C01823=1018.796,230.980,371.499,168.951,51.014,159.703
C01824=1018.803,231.229,371.472,168.955,51.007,159.702
C01825=1018.808,231.478,371.446,168.959,51.001,159.701
C01826=1018.814,231.727,371.419,168.964,50.995,159.701
C01827=1018.820,231.975,371.392,168.967,50.989,159.700
C01828=1018.826,232.223,371.365,168.971,50.983,159.699
C01829=1018.832,232.472,371.338,168.976,50.976,159.699
C01830=1018.838,232.720,371.311,168.979,50.970,159.698
C01831=1018.844,232.969,371.285,168.984,50.964,159.698
C01832=1018.850,233.217,371.258,168.988,50.958,159.697
C01833=1018.856,233.444,371.234,168.992,50.952,159.697
C01834=1018.861,233.670,371.210,168.996,50.947,159.696
C01835=1018.867,233.895,371.185,169.000,50.941,159.695
C01836=1018.872,234.122,371.161,169.003,50.936,159.695
C01837=1018.877,234.348,371.136,169.007,50.930,159.694
C01838=1018.882,234.574,371.112,169.011,50.924,159.694
C01839=1018.888,234.800,371.087,169.015,50.919,159.693
C01840=1018.893,235.026,371.063,169.019,50.913,159.693
C01841=1018.900,235.275,371.036,169.022,50.907,159.692
C01842=1018.905,235.523,371.009,169.027,50.901,159.692
C01843=1018.911,235.771,370.982,169.031,50.895,159.691
C01844=1018.917,236.019,370.955,169.034,50.889,159.690
C01845=1018.924,236.268,370.928,169.040,50.883,159.690
C01846=1018.929,236.517,370.902,169.043,50.877,159.689
C01847=1018.936,236.766,370.875,169.047,50.871,159.688
C01848=1018.942,237.014,370.847,169.052,50.864,159.688
C01849=1018.948,237.262,370.821,169.056,50.859,159.687
C01850=1018.954,237.511,370.794,169.060,50.852,159.687
C01851=1018.960,237.759,370.766,169.064,50.846,159.686
C01852=1018.966,238.007,370.740,169.068,50.840,159.686
C01853=1018.972,238.256,370.713,169.073,50.834,159.685
C01854=1018.978,238.504,370.686,169.077,50.828,159.684
C01855=1018.985,238.753,370.658,169.080,50.822,159.684
C01856=1018.990,239.002,370.631,169.085,50.817,159.683
C01857=1018.996,239.249,370.604,169.089,50.810,159.683
C01858=1019.002,239.498,370.577,169.093,50.805,159.682
C01859=1019.008,239.747,370.550,169.098,50.799,159.682
C01860=1019.014,239.996,370.522,169.102,50.793,159.681
C01861=1019.020,240.244,370.495,169.106,50.787,159.681
C01862=1019.026,240.492,370.468,169.111,50.781,159.680
C01863=1019.032,240.740,370.439,169.114,50.775,159.680
C01864=1019.037,240.989,370.413,169.119,50.770,159.679
C01865=1019.044,241.237,370.385,169.123,50.764,159.678
C01866=1019.049,241.486,370.358,169.127,50.758,159.678
C01867=1019.056,241.734,370.330,169.131,50.752,159.677
C01868=1019.061,241.983,370.303,169.135,50.747,159.677
C01869=1019.067,242.231,370.275,169.140,50.741,159.676
C01870=1019.073,242.480,370.248,169.144,50.735,159.676
C01871=1019.079,242.728,370.220,169.148,50.730,159.675
C01872=1019.085,242.976,370.193,169.153,50.723,159.675
C01873=1019.091,243.225,370.166,169.157,50.718,159.674
C01874=1019.097,243.473,370.138,169.161,50.712,159.674
C01875=1019.102,243.721,370.110,169.165,50.707,159.673
C01876=1019.109,243.970,370.082,169.170,50.701,159.673
C01877=1019.114,244.218,370.054,169.174,50.695,159.672
C01878=1019.121,244.467,370.027,169.178,50.690,159.672
C01879=1019.126,244.715,369.999,169.182,50.684,159.671
C01880=1019.132,244.964,369.971,169.187,50.679,159.671
C01881=1019.138,245.211,369.943,169.191,50.673,159.670
C01882=1019.144,245.460,369.915,169.195,50.667,159.670
C01883=1019.149,245.708,369.887,169.199,50.662,159.669
C01884=1019.156,245.957,369.860,169.203,50.657,159.669
C01885=1019.161,246.205,369.832,169.208,50.651,159.669
C01886=1019.168,246.454,369.804,169.213,50.645,159.668
C01887=1019.174,246.703,369.776,169.217,50.640,159.668
C01888=1019.179,246.951,369.748,169.221,50.635,159.667
C01889=1019.186,247.199,369.720,169.226,50.628,159.667
C01890=1019.191,247.447,369.692,169.230,50.623,159.666
C01891=1019.197,247.696,369.664,169.234,50.618,159.666
C01892=1019.203,247.944,369.637,169.238,50.612,159.665
C01893=1019.208,248.167,369.611,169.242,50.608,159.665
C01894=1019.213,248.390,369.587,169.245,50.602,159.664
C01895=1019.219,248.612,369.562,169.250,50.598,159.664
C01896=1019.224,248.835,369.536,169.253,50.593,159.663
C01897=1019.230,249.058,369.511,169.258,50.588,159.663
C01898=1019.235,249.280,369.486,169.262,50.583,159.663
C01899=1019.241,249.504,369.461,169.265,50.578,159.662
C01900=1019.246,249.726,369.436,169.269,50.573,159.662
C01901=1019.252,249.975,369.408,169.273,50.568,159.661
C01902=1019.258,250.224,369.380,169.278,50.562,159.661
C01903=1019.264,250.472,369.352,169.282,50.557,159.660
C01904=1019.271,250.720,369.323,169.287,50.551,159.660
C01905=1019.276,250.968,369.295,169.291,50.546,159.660
C01906=1019.282,251.216,369.267,169.295,50.541,159.659
C01907=1019.288,251.465,369.239,169.300,50.536,159.659
C01908=1019.294,251.714,369.211,169.305,50.530,159.659
C01909=1019.300,251.962,369.183,169.309,50.525,159.658
C01910=1019.306,252.210,369.155,169.313,50.519,159.658
C01911=1019.312,252.459,369.127,169.317,50.514,159.657
C01912=1019.319,252.707,369.098,169.321,50.509,159.657
C01913=1019.325,252.955,369.070,169.326,50.503,159.656
C01914=1019.331,253.203,369.042,169.331,50.498,159.656
C01915=1019.337,253.452,369.014,169.335,50.493,159.656
C01916=1019.344,253.700,368.986,169.339,50.488,159.655
C01917=1019.350,253.949,368.957,169.343,50.482,159.655
C01918=1019.356,254.196,368.930,169.348,50.477,159.654
C01919=1019.362,254.445,368.902,169.352,50.471,159.654
C01920=1019.368,254.693,368.872,169.357,50.466,159.653
C01921=1019.375,254.942,368.845,169.361,50.461,159.653
C01922=1019.380,255.191,368.816,169.366,50.455,159.653
C01923=1019.386,255.439,368.788,169.370,50.450,159.652
C01924=1019.393,255.686,368.760,169.375,50.445,159.652
C01925=1019.399,255.935,368.732,169.379,50.440,159.651
C01926=1019.405,256.184,368.703,169.383,50.435,159.651
C01927=1019.412,256.432,368.675,169.388,50.429,159.650
C01928=1019.418,256.680,368.647,169.393,50.424,159.650
C01929=1019.423,256.929,368.619,169.397,50.419,159.650
C01930=1019.430,257.176,368.590,169.401,50.414,159.649
C01931=1019.436,257.425,368.562,169.406,50.409,159.649
C01932=1019.442,257.673,368.533,169.411,50.403,159.649
C01933=1019.449,257.922,368.505,169.415,50.398,159.648
C01934=1019.455,258.170,368.476,169.419,50.393,159.648
C01935=1019.461,258.419,368.448,169.423,50.388,159.647
C01936=1019.468,258.667,368.420,169.429,50.383,159.647
C01937=1019.474,258.915,368.391,169.433,50.378,159.647
C01938=1019.480,259.164,368.363,169.437,50.372,159.646
C01939=1019.487,259.412,368.334,169.442,50.368,159.646
C01940=1019.492,259.660,368.306,169.446,50.362,159.645
C01941=1019.498,259.908,368.277,169.451,50.357,159.645
C01942=1019.505,260.156,368.248,169.456,50.352,159.645
C01943=1019.511,260.405,368.220,169.460,50.347,159.645
C01944=1019.517,260.653,368.191,169.464,50.342,159.644
C01945=1019.523,260.901,368.162,169.469,50.337,159.644
C01946=1019.529,261.149,368.133,169.473,50.333,159.644
C01947=1019.535,261.398,368.104,169.477,50.327,159.643
C01948=1019.542,261.646,368.075,169.482,50.323,159.643
C01949=1019.548,261.894,368.046,169.487,50.318,159.643
C01950=1019.554,262.142,368.017,169.492,50.313,159.642
C01951=1019.560,262.390,367.988,169.496,50.308,159.642
C01952=1019.566,262.639,367.960,169.501,50.303,159.642
C01953=1019.571,262.861,367.934,169.504,50.299,159.641
C01954=1019.577,263.083,367.908,169.509,50.294,159.641
C01955=1019.582,263.305,367.882,169.513,50.290,159.641
C01956=1019.588,263.527,367.856,169.517,50.286,159.641
C01957=1019.593,263.749,367.830,169.521,50.281,159.640
C01958=1019.599,263.970,367.804,169.525,50.277,159.640
C01959=1019.605,264.192,367.778,169.529,50.272,159.639
C01960=1019.610,264.415,367.752,169.534,50.268,159.639
C01961=1019.616,264.663,367.723,169.538,50.263,159.639
C01962=1019.622,264.911,367.694,169.542,50.259,159.639
C01963=1019.629,265.159,367.665,169.547,50.254,159.638
C01964=1019.635,265.407,367.636,169.551,50.249,159.638
C01965=1019.640,265.656,367.606,169.556,50.245,159.638
C01966=1019.647,265.904,367.577,169.560,50.240,159.638
C01967=1019.653,266.152,367.548,169.566,50.235,159.637
C01968=1019.659,266.400,367.519,169.570,50.230,159.637
C01969=1019.665,266.648,367.490,169.575,50.226,159.637
C01970=1019.671,266.896,367.460,169.579,50.221,159.637
C01971=1019.678,267.145,367.430,169.584,50.216,159.636
C01972=1019.684,267.393,367.401,169.589,50.212,159.636
C01973=1019.691,267.641,367.372,169.593,50.207,159.636
C01974=1019.696,267.890,367.343,169.598,50.202,159.635
C01975=1019.702,268.138,367.314,169.602,50.198,159.635
C01976=1019.709,268.385,367.284,169.607,50.193,159.635
C01977=1019.714,268.634,367.254,169.612,50.188,159.635
C01978=1019.721,268.882,367.225,169.617,50.183,159.634
C01979=1019.727,269.131,367.196,169.621,50.179,159.634
C01980=1019.734,269.379,367.167,169.626,50.174,159.634
C01981=1019.740,269.627,367.136,169.630,50.170,159.634
C01982=1019.746,269.875,367.107,169.635,50.165,159.633
C01983=1019.751,270.123,367.078,169.639,50.160,159.633
C01984=1019.758,270.371,367.048,169.644,50.156,159.633
C01985=1019.765,270.619,367.019,169.649,50.152,159.633
C01986=1019.770,270.867,366.988,169.653,50.147,159.632
C01987=1019.777,271.115,366.959,169.658,50.142,159.632
C01988=1019.782,271.364,366.930,169.662,50.138,159.632
C01989=1019.789,271.611,366.900,169.668,50.133,159.632
C01990=1019.796,271.860,366.870,169.673,50.129,159.632
C01991=1019.801,272.108,366.840,169.677,50.124,159.631
C01992=1019.808,272.356,366.811,169.682,50.120,159.631
C01993=1019.814,272.604,366.781,169.687,50.116,159.631
C01994=1019.820,272.853,366.751,169.691,50.111,159.631
C01995=1019.826,273.101,366.721,169.696,50.106,159.630
C01996=1019.832,273.349,366.692,169.701,50.102,159.630
C01997=1019.838,273.597,366.661,169.705,50.098,159.630
C01998=1019.845,273.845,366.632,169.710,50.093,159.630
C01999=1019.851,274.093,366.602,169.715,50.089,159.630
C02000=1019.857,274.341,366.572,169.719,50.085,159.629
C02001=1019.864,274.590,366.542,169.724,50.081,159.629
C02002=1019.870,274.837,366.512,169.729,50.076,159.629
C02003=1019.876,275.086,366.483,169.733,50.071,159.629
C02004=1019.882,275.333,366.453,169.739,50.067,159.629
C02005=1019.889,275.582,366.422,169.744,50.062,159.628
C02006=1019.895,275.830,366.393,169.749,50.058,159.628
C02007=1019.901,276.078,366.363,169.753,50.054,159.628
C02008=1019.907,276.326,366.332,169.758,50.050,159.628
C02009=1019.914,276.574,366.302,169.763,50.045,159.628
C02010=1019.920,276.823,366.272,169.768,50.041,159.628
C02011=1019.926,277.071,366.242,169.772,50.037,159.627
C02012=1019.932,277.318,366.212,169.777,50.033,159.627
C02013=1019.938,277.542,366.184,169.781,50.029,159.627
C02014=1019.943,277.767,366.157,169.786,50.025,159.627
C02015=1019.949,277.991,366.130,169.790,50.021,159.627
C02016=1019.955,278.215,366.102,169.795,50.017,159.627
C02017=1019.960,278.440,366.075,169.799,50.014,159.627
C02018=1019.966,278.664,366.047,169.804,50.010,159.626
C02019=1019.971,278.888,366.020,169.808,50.006,159.626
C02020=1019.977,279.112,365.993,169.813,50.002,159.626
C02021=1019.983,279.361,365.962,169.817,49.998,159.626
C02022=1019.990,279.608,365.932,169.822,49.994,159.626
C02023=1019.996,279.857,365.901,169.827,49.990,159.626
C02024=1020.002,280.105,365.871,169.832,49.986,159.626
C02025=1020.008,280.353,365.840,169.837,49.982,159.626
C02026=1020.014,280.601,365.810,169.841,49.977,159.625
C02027=1020.021,280.849,365.780,169.846,49.973,159.625
C02028=1020.027,281.097,365.750,169.851,49.969,159.625
C02029=1020.033,281.345,365.719,169.856,49.965,159.625
C02030=1020.039,281.593,365.689,169.861,49.961,159.625
C02031=1020.046,281.841,365.659,169.866,49.957,159.625
C02032=1020.053,282.089,365.627,169.870,49.953,159.625
C02033=1020.058,282.337,365.597,169.875,49.949,159.624
C02034=1020.065,282.585,365.566,169.880,49.945,159.624
C02035=1020.071,282.834,365.536,169.885,49.941,159.624
C02036=1020.078,283.081,365.506,169.890,49.937,159.624
C02037=1020.084,283.330,365.475,169.895,49.933,159.624
C02038=1020.090,283.577,365.444,169.900,49.929,159.624
C02039=1020.097,283.825,365.413,169.906,49.924,159.624
C02040=1020.103,284.073,365.384,169.910,49.920,159.624
C02041=1020.110,284.321,365.353,169.915,49.916,159.624
C02042=1020.117,284.569,365.321,169.920,49.912,159.624
C02043=1020.122,284.817,365.291,169.925,49.909,159.623
C02044=1020.129,285.066,365.260,169.930,49.905,159.623
C02045=1020.135,285.313,365.229,169.935,49.901,159.623
C02046=1020.141,285.561,365.199,169.940,49.897,159.623
C02047=1020.147,285.809,365.167,169.945,49.893,159.623
C02048=1020.154,286.057,365.137,169.950,49.889,159.623
C02049=1020.161,286.305,365.105,169.955,49.886,159.623
C02050=1020.166,286.553,365.075,169.960,49.882,159.623
C02051=1020.173,286.801,365.044,169.965,49.878,159.623
C02052=1020.180,287.049,365.013,169.970,49.874,159.623
C02053=1020.186,287.296,364.982,169.975,49.870,159.623
C02054=1020.192,287.545,364.951,169.980,49.866,159.623
C02055=1020.199,287.793,364.920,169.985,49.863,159.623
C02056=1020.205,288.041,364.889,169.990,49.859,159.623
C02057=1020.211,288.289,364.858,169.995,49.855,159.623
C02058=1020.218,288.537,364.827,170.000,49.851,159.623
C02059=1020.224,288.784,364.796,170.005,49.847,159.623
C02060=1020.231,289.032,364.765,170.010,49.844,159.623
C02061=1020.237,289.281,364.734,170.015,49.840,159.622
C02062=1020.244,289.529,364.702,170.020,49.836,159.623
C02063=1020.250,289.776,364.671,170.025,49.832,159.622
C02064=1020.256,290.025,364.640,170.031,49.828,159.622
C02065=1020.262,290.273,364.609,170.036,49.824,159.622
C02066=1020.269,290.521,364.577,170.041,49.821,159.622
C02067=1020.275,290.768,364.546,170.046,49.817,159.622
C02068=1020.282,291.016,364.515,170.052,49.814,159.622
C02069=1020.288,291.264,364.484,170.057,49.810,159.622
C02070=1020.295,291.512,364.453,170.061,49.806,159.622
C02071=1020.302,291.760,364.421,170.067,49.803,159.622
C02072=1020.307,292.007,364.389,170.072,49.799,159.622
C02073=1020.314,292.238,364.361,170.076,49.796,159.622
C02074=1020.320,292.469,364.331,170.081,49.792,159.622
C02075=1020.325,292.699,364.302,170.086,49.788,159.622
C02076=1020.332,292.929,364.273,170.091,49.786,159.622
C02077=1020.338,293.160,364.243,170.096,49.782,159.622
C02078=1020.343,293.390,364.214,170.101,49.778,159.622
C02079=1020.349,293.620,364.185,170.105,49.775,159.622
C02080=1020.355,293.851,364.155,170.110,49.772,159.623
C02081=1020.361,294.098,364.123,170.116,49.769,159.623
C02082=1020.367,294.346,364.092,170.121,49.765,159.623
C02083=1020.373,294.595,364.060,170.126,49.762,159.623
C02084=1020.380,294.842,364.028,170.131,49.758,159.623
C02085=1020.386,295.090,363.996,170.136,49.755,159.623
C02086=1020.392,295.338,363.963,170.141,49.751,159.623
C02087=1020.399,295.585,363.932,170.147,49.748,159.623
C02088=1020.405,295.834,363.900,170.152,49.745,159.623
C02089=1020.412,296.081,363.868,170.157,49.741,159.623
C02090=1020.418,296.329,363.836,170.163,49.738,159.623
C02091=1020.424,296.577,363.805,170.168,49.734,159.623
C02092=1020.431,296.825,363.772,170.173,49.731,159.623
C02093=1020.437,297.073,363.740,170.178,49.728,159.623
C02094=1020.443,297.321,363.709,170.183,49.724,159.623
C02095=1020.450,297.568,363.676,170.189,49.721,159.623
C02096=1020.456,297.816,363.644,170.194,49.718,159.624
C02097=1020.462,298.064,363.612,170.199,49.714,159.623
C02098=1020.469,298.312,363.580,170.204,49.711,159.624
C02099=1020.475,298.560,363.548,170.210,49.707,159.624
C02100=1020.482,298.808,363.515,170.215,49.704,159.624
C02101=1020.488,299.055,363.484,170.220,49.701,159.624
C02102=1020.495,299.303,363.451,170.226,49.698,159.624
C02103=1020.501,299.551,363.420,170.231,49.694,159.624
C02104=1020.507,299.799,363.388,170.236,49.691,159.624
C02105=1020.514,300.047,363.355,170.241,49.688,159.624
C02106=1020.521,300.294,363.323,170.247,49.685,159.624
C02107=1020.527,300.542,363.291,170.252,49.681,159.624
C02108=1020.534,300.790,363.259,170.257,49.678,159.625
C02109=1020.540,301.038,363.227,170.263,49.675,159.625
C02110=1020.547,301.285,363.195,170.268,49.671,159.625
C02111=1020.553,301.533,363.163,170.273,49.668,159.625
C02112=1020.559,301.781,363.130,170.279,49.665,159.625
C02113=1020.567,302.029,363.097,170.284,49.662,159.625
C02114=1020.573,302.277,363.065,170.289,49.658,159.625
C02115=1020.580,302.524,363.033,170.295,49.656,159.625
C02116=1020.586,302.772,363.000,170.300,49.653,159.626
C02117=1020.592,303.020,362.968,170.305,49.649,159.626
C02118=1020.599,303.267,362.936,170.311,49.646,159.626
C02119=1020.606,303.516,362.903,170.317,49.642,159.626
C02120=1020.613,303.763,362.871,170.322,49.639,159.626
C02121=1020.619,304.011,362.839,170.328,49.637,159.626
C02122=1020.625,304.259,362.806,170.333,49.633,159.626
C02123=1020.632,304.506,362.774,170.339,49.630,159.627
C02124=1020.639,304.754,362.741,170.344,49.627,159.627
C02125=1020.646,305.002,362.709,170.349,49.624,159.627
C02126=1020.652,305.250,362.677,170.355,49.621,159.627
C02127=1020.658,305.497,362.644,170.360,49.618,159.627
C02128=1020.666,305.745,362.611,170.365,49.614,159.627
C02129=1020.672,305.993,362.579,170.371,49.612,159.628
C02130=1020.679,306.240,362.547,170.377,49.608,159.628
C02131=1020.686,306.489,362.513,170.383,49.605,159.628
C02132=1020.693,306.736,362.481,170.388,49.602,159.628
C02133=1020.699,306.976,362.450,170.394,49.599,159.628
C02134=1020.706,307.214,362.418,170.399,49.596,159.628
C02135=1020.712,307.454,362.387,170.404,49.594,159.628
C02136=1020.719,307.693,362.355,170.409,49.590,159.629
C02137=1020.725,307.932,362.324,170.415,49.588,159.629
C02138=1020.732,308.171,362.292,170.420,49.584,159.629
C02139=1020.739,308.410,362.261,170.426,49.582,159.629
C02140=1020.745,308.650,362.229,170.431,49.579,159.629
C02141=1020.752,308.897,362.196,170.437,49.576,159.630
C02142=1020.759,309.144,362.164,170.442,49.573,159.630
C02143=1020.766,309.393,362.131,170.447,49.569,159.630
C02144=1020.773,309.640,362.098,170.454,49.567,159.630
C02145=1020.780,309.888,362.065,170.459,49.563,159.630
C02146=1020.786,310.135,362.032,170.465,49.561,159.631
C02147=1020.792,310.383,361.999,170.470,49.558,159.631
C02148=1020.800,310.631,361.965,170.476,49.555,159.631
C02149=1020.806,310.878,361.933,170.481,49.552,159.631
C02150=1020.812,311.125,361.899,170.487,49.550,159.632
C02151=1020.819,311.374,361.865,170.493,49.547,159.632
C02152=1020.825,311.621,361.832,170.498,49.544,159.632
C02153=1020.832,311.869,361.799,170.504,49.542,159.632
C02154=1020.838,312.116,361.765,170.509,49.539,159.633
C02155=1020.845,312.365,361.732,170.515,49.536,159.633
C02156=1020.852,312.612,361.698,170.521,49.533,159.633
C02157=1020.858,312.859,361.665,170.526,49.531,159.633
C02158=1020.865,313.107,361.632,170.532,49.528,159.634
C02159=1020.871,313.354,361.598,170.538,49.526,159.634
C02160=1020.878,313.602,361.565,170.544,49.523,159.634
C02161=1020.884,313.849,361.531,170.550,49.520,159.635
C02162=1020.892,314.097,361.497,170.556,49.517,159.635
C02163=1020.898,314.345,361.463,170.561,49.515,159.635
C02164=1020.904,314.593,361.430,170.567,49.512,159.636
C02165=1020.912,314.840,361.396,170.573,49.510,159.636
C02166=1020.918,315.087,361.363,170.578,49.507,159.636
C02167=1020.924,315.336,361.329,170.584,49.504,159.636
C02168=1020.931,315.583,361.296,170.590,49.502,159.637
C02169=1020.938,315.831,361.262,170.595,49.499,159.637
C02170=1020.945,316.078,361.228,170.601,49.497,159.637
C02171=1020.951,316.325,361.194,170.608,49.494,159.638
C02172=1020.958,316.573,361.160,170.613,49.491,159.638
C02173=1020.965,316.821,361.127,170.619,49.488,159.638
C02174=1020.971,317.069,361.093,170.625,49.486,159.639
C02175=1020.978,317.316,361.059,170.630,49.483,159.639
C02176=1020.986,317.564,361.025,170.636,49.481,159.639
C02177=1020.992,317.811,360.992,170.642,49.478,159.639
C02178=1020.999,318.059,360.957,170.649,49.476,159.640
C02179=1021.006,318.307,360.924,170.655,49.473,159.640
C02180=1021.013,318.554,360.890,170.660,49.471,159.641
C02181=1021.020,318.801,360.856,170.666,49.468,159.641
C02182=1021.026,319.049,360.822,170.672,49.465,159.641
C02183=1021.033,319.297,360.788,170.678,49.463,159.642
C02184=1021.040,319.545,360.754,170.683,49.461,159.642
C02185=1021.046,319.792,360.720,170.690,49.458,159.642
C02186=1021.054,320.040,360.686,170.696,49.456,159.643
C02187=1021.061,320.287,360.653,170.702,49.453,159.643
C02188=1021.068,320.534,360.618,170.707,49.451,159.643
C02189=1021.075,320.782,360.584,170.713,49.448,159.644
C02190=1021.082,321.030,360.550,170.719,49.446,159.644
C02191=1021.088,321.277,360.516,170.726,49.443,159.644
C02192=1021.096,321.525,360.482,170.732,49.441,159.645
C02193=1021.102,321.767,360.449,170.737,49.439,159.645
C02194=1021.109,322.008,360.415,170.743,49.436,159.645
C02195=1021.116,322.250,360.382,170.749,49.434,159.646
C02196=1021.123,322.492,360.349,170.755,49.432,159.646
C02197=1021.130,322.733,360.315,170.761,49.430,159.647
C02198=1021.137,322.975,360.282,170.766,49.427,159.647
C02199=1021.144,323.217,360.249,170.772,49.425,159.647
C02200=1021.151,323.458,360.215,170.778,49.423,159.648
C02201=1021.158,323.706,360.181,170.785,49.420,159.648
C02202=1021.164,323.954,360.147,170.791,49.418,159.649
C02203=1021.172,324.201,360.112,170.797,49.416,159.649
C02204=1021.179,324.448,360.078,170.802,49.413,159.649
C02205=1021.186,324.696,360.043,170.809,49.411,159.650
C02206=1021.193,324.944,360.009,170.815,49.408,159.650
C02207=1021.201,325.192,359.975,170.821,49.406,159.651
C02208=1021.207,325.439,359.940,170.827,49.404,159.651
C02209=1021.215,325.687,359.906,170.834,49.401,159.652
C02210=1021.222,325.934,359.872,170.840,49.399,159.652
C02211=1021.229,326.182,359.838,170.846,49.397,159.652
C02212=1021.236,326.429,359.803,170.852,49.395,159.653
C02213=1021.244,326.676,359.768,170.859,49.393,159.653
C02214=1021.250,326.924,359.734,170.865,49.391,159.654
C02215=1021.258,327.171,359.699,170.870,49.388,159.654
C02216=1021.264,327.418,359.664,170.876,49.386,159.655
C02217=1021.272,327.667,359.629,170.882,49.384,159.655
C02218=1021.278,327.914,359.594,170.889,49.382,159.656
C02219=1021.286,328.162,359.560,170.895,49.380,159.656
C02220=1021.292,328.409,359.525,170.902,49.378,159.657
C02221=1021.299,328.656,359.489,170.908,49.376,159.657
C02222=1021.306,328.904,359.454,170.915,49.374,159.658
C02223=1021.313,329.151,359.420,170.921,49.372,159.658
C02224=1021.321,329.399,359.384,170.927,49.370,159.659
C02225=1021.328,329.646,359.349,170.933,49.368,159.659
C02226=1021.334,329.894,359.314,170.940,49.366,159.660
C02227=1021.342,330.141,359.280,170.946,49.364,159.660
C02228=1021.349,330.388,359.244,170.952,49.362,159.661
C02229=1021.356,330.636,359.209,170.958,49.360,159.661
C02230=1021.363,330.883,359.174,170.965,49.357,159.662
C02231=1021.370,331.130,359.139,170.971,49.355,159.662
C02232=1021.378,331.378,359.104,170.977,49.354,159.663
C02233=1021.384,331.626,359.069,170.983,49.352,159.663
C02234=1021.392,331.873,359.033,170.990,49.350,159.664
C02235=1021.399,332.120,358.998,170.996,49.348,159.664
C02236=1021.406,332.368,358.963,171.002,49.346,159.665
C02237=1021.413,332.615,358.928,171.009,49.344,159.665
C02238=1021.421,332.863,358.892,171.015,49.342,159.666
C02239=1021.428,333.110,358.857,171.022,49.340,159.666
C02240=1021.435,333.357,358.822,171.028,49.339,159.667
C02241=1021.442,333.605,358.786,171.035,49.336,159.668
C02242=1021.450,333.852,358.750,171.041,49.335,159.668
C02243=1021.456,334.099,358.715,171.047,49.333,159.669
C02244=1021.464,334.347,358.679,171.054,49.331,159.669
C02245=1021.471,334.594,358.644,171.061,49.329,159.670
C02246=1021.478,334.841,358.608,171.067,49.327,159.670
C02247=1021.485,335.089,358.572,171.074,49.326,159.671
C02248=1021.492,335.335,358.537,171.080,49.324,159.672
C02249=1021.500,335.584,358.501,171.087,49.322,159.672
C02250=1021.507,335.830,358.465,171.094,49.320,159.673
C02251=1021.514,336.078,358.430,171.100,49.319,159.674
C02252=1021.521,336.325,358.394,171.106,49.317,159.674
C02253=1021.528,336.565,358.358,171.112,49.316,159.675
C02254=1021.535,336.805,358.324,171.118,49.314,159.675
C02255=1021.542,337.044,358.289,171.126,49.312,159.676
C02256=1021.549,337.283,358.254,171.132,49.310,159.676
C02257=1021.556,337.523,358.220,171.138,49.309,159.677
C02258=1021.563,337.763,358.185,171.144,49.307,159.678
C02259=1021.570,338.002,358.151,171.151,49.305,159.678
C02260=1021.578,338.242,358.115,171.157,49.304,159.679
C02261=1021.585,338.488,358.080,171.164,49.302,159.679
C02262=1021.592,338.736,358.044,171.170,49.301,159.680
C02263=1021.599,338.983,358.008,171.178,49.299,159.681
C02264=1021.607,339.231,357.972,171.184,49.297,159.681
C02265=1021.615,339.478,357.936,171.190,49.296,159.682
C02266=1021.622,339.725,357.900,171.198,49.294,159.683
C02267=1021.629,339.972,357.864,171.204,49.293,159.683
C02268=1021.636,340.220,357.827,171.210,49.291,159.684
C02269=1021.643,340.467,357.791,171.218,49.290,159.685
C02270=1021.651,340.714,357.755,171.224,49.288,159.685
C02271=1021.659,340.962,357.719,171.231,49.286,159.686
C02272=1021.665,341.209,357.682,171.238,49.285,159.687
C02273=1021.673,341.456,357.646,171.244,49.283,159.687
C02274=1021.680,341.704,357.610,171.251,49.282,159.688
C02275=1021.688,341.950,357.573,171.258,49.280,159.689
C02276=1021.695,342.197,357.536,171.265,49.279,159.690
C02277=1021.702,342.445,357.500,171.271,49.277,159.690
C02278=1021.710,342.692,357.464,171.279,49.276,159.691
C02279=1021.717,342.940,357.427,171.285,49.274,159.692
C02280=1021.724,343.186,357.391,171.292,49.273,159.692
C02281=1021.732,343.434,357.354,171.299,49.271,159.693
C02282=1021.739,343.681,357.318,171.306,49.271,159.694
C02283=1021.747,343.928,357.281,171.313,49.269,159.695
C02284=1021.755,344.176,357.244,171.320,49.268,159.695
C02285=1021.762,344.423,357.207,171.327,49.266,159.696
C02286=1021.769,344.670,357.171,171.333,49.265,159.697
C02287=1021.777,344.917,357.135,171.341,49.263,159.698
C02288=1021.784,345.164,357.097,171.347,49.262,159.698
C02289=1021.792,345.412,357.061,171.354,49.261,159.699
C02290=1021.799,345.659,357.024,171.361,49.259,159.700
C02291=1021.806,345.906,356.987,171.368,49.258,159.701
C02292=1021.814,346.153,356.950,171.375,49.257,159.701
C02293=1021.822,346.400,356.913,171.382,49.256,159.702
C02294=1021.829,346.648,356.877,171.389,49.254,159.703
C02295=1021.837,346.894,356.840,171.396,49.253,159.704
C02296=1021.844,347.142,356.803,171.403,49.252,159.705
C02297=1021.852,347.389,356.766,171.411,49.251,159.705
C02298=1021.859,347.636,356.728,171.417,49.249,159.706
C02299=1021.867,347.883,356.692,171.425,49.248,159.707
C02300=1021.874,348.131,356.655,171.431,49.247,159.708
C02301=1021.882,348.378,356.618,171.439,49.245,159.708
C02302=1021.890,348.625,356.580,171.446,49.245,159.709
C02303=1021.898,348.871,356.543,171.453,49.244,159.710
C02304=1021.905,349.119,356.506,171.460,49.242,159.711
C02305=1021.912,349.366,356.468,171.467,49.241,159.712
C02306=1021.920,349.613,356.431,171.474,49.240,159.713
C02307=1021.927,349.860,356.394,171.482,49.239,159.714
C02308=1021.935,350.108,356.356,171.488,49.238,159.714
C02309=1021.943,350.354,356.319,171.496,49.237,159.715
C02310=1021.950,350.601,356.281,171.503,49.236,159.716
C02311=1021.958,350.848,356.245,171.510,49.235,159.717
C02312=1021.966,351.095,356.207,171.518,49.234,159.718
C02313=1021.973,351.333,356.171,171.524,49.232,159.719
C02314=1021.981,351.571,356.135,171.531,49.232,159.719
C02315=1021.988,351.809,356.098,171.539,49.231,159.720
C02316=1021.995,352.047,356.062,171.546,49.230,159.721
C02317=1022.003,352.286,356.026,171.552,49.229,159.722
C02318=1022.010,352.524,355.990,171.560,49.228,159.723
C02319=1022.018,352.761,355.954,171.566,49.227,159.724
C02320=1022.026,352.999,355.917,171.574,49.226,159.725
C02321=1022.033,353.246,355.880,171.581,49.225,159.726
C02322=1022.040,353.493,355.842,171.589,49.224,159.727
C02323=1022.049,353.740,355.804,171.596,49.222,159.727
C02324=1022.056,353.987,355.767,171.603,49.222,159.728
C02325=1022.064,354.234,355.729,171.610,49.221,159.729
C02326=1022.072,354.481,355.691,171.619,49.220,159.730
C02327=1022.080,354.728,355.653,171.625,49.220,159.731
C02328=1022.088,354.976,355.615,171.633,49.219,159.732
C02329=1022.095,355.222,355.577,171.641,49.218,159.733
C02330=1022.103,355.469,355.539,171.648,49.217,159.734
C02331=1022.111,355.716,355.501,171.655,49.216,159.735
C02332=1022.119,355.963,355.463,171.663,49.215,159.736
C02333=1022.127,356.210,355.425,171.670,49.215,159.737
C02334=1022.134,356.457,355.387,171.678,49.214,159.738
C02335=1022.142,356.704,355.349,171.686,49.213,159.739
C02336=1022.150,356.951,355.310,171.692,49.212,159.740
C02337=1022.158,357.198,355.273,171.700,49.211,159.741
C02338=1022.166,357.445,355.235,171.708,49.210,159.742
C02339=1022.174,357.692,355.196,171.716,49.209,159.743
C02340=1022.182,357.939,355.158,171.723,49.209,159.744
C02341=1022.190,358.186,355.119,171.731,49.208,159.745
C02342=1022.198,358.432,355.081,171.739,49.207,159.746
C02343=1022.206,358.680,355.042,171.747,49.207,159.747
C02344=1022.213,358.926,355.004,171.753,49.206,159.748
C02345=1022.221,359.173,354.965,171.761,49.206,159.749
C02346=1022.230,359.420,354.928,171.769,49.205,159.750
C02347=1022.238,359.667,354.889,171.777,49.204,159.751
C02348=1022.246,359.914,354.851,171.785,49.203,159.752
C02349=1022.254,360.161,354.812,171.792,49.203,159.753
C02350=1022.261,360.408,354.773,171.800,49.202,159.754
C02351=1022.269,360.655,354.735,171.808,49.201,159.755
C02352=1022.277,360.901,354.696,171.816,49.201,159.756
C02353=1022.285,361.148,354.657,171.823,49.200,159.757
C02354=1022.293,361.396,354.618,171.831,49.200,159.758
C02355=1022.301,361.642,354.579,171.839,49.199,159.759
C02356=1022.309,361.889,354.540,171.847,49.199,159.760
C02357=1022.317,362.136,354.502,171.855,49.199,159.762
C02358=1022.325,362.382,354.463,171.863,49.198,159.762
C02359=1022.333,362.629,354.424,171.870,49.197,159.764
C02360=1022.341,362.876,354.385,171.878,49.197,159.765
C02361=1022.349,363.123,354.346,171.886,49.197,159.766
C02362=1022.357,363.370,354.306,171.894,49.196,159.767
C02363=1022.365,363.617,354.268,171.902,49.196,159.768
C02364=1022.373,363.863,354.229,171.911,49.195,159.769
C02365=1022.381,364.110,354.190,171.919,49.195,159.770
C02366=1022.390,364.357,354.151,171.926,49.195,159.771
C02367=1022.398,364.604,354.111,171.934,49.194,159.773
C02368=1022.406,364.851,354.072,171.942,49.194,159.774
C02369=1022.414,365.098,354.033,171.950,49.193,159.775
C02370=1022.422,365.344,353.994,171.958,49.193,159.776
C02371=1022.431,365.592,353.955,171.966,49.192,159.777
C02372=1022.438,365.837,353.916,171.974,49.192,159.778
C02373=1022.447,366.079,353.877,171.982,49.192,159.779
C02374=1022.455,366.321,353.839,171.991,49.191,159.781
C02375=1022.463,366.562,353.800,171.999,49.191,159.782
C02376=1022.471,366.804,353.762,172.006,49.191,159.783
C02377=1022.479,367.044,353.723,172.014,49.190,159.784
C02378=1022.487,367.286,353.685,172.022,49.190,159.785
C02379=1022.495,367.528,353.646,172.030,49.190,159.786
C02380=1022.504,367.769,353.607,172.039,49.189,159.788
C02381=1022.512,368.015,353.568,172.047,49.189,159.789
C02382=1022.520,368.262,353.528,172.055,49.189,159.790
C02383=1022.529,368.509,353.489,172.063,49.189,159.791
C02384=1022.536,368.756,353.449,172.072,49.189,159.793
C02385=1022.545,369.002,353.410,172.080,49.188,159.794
C02386=1022.553,369.249,353.369,172.088,49.188,159.795
C02387=1022.562,369.496,353.329,172.096,49.188,159.796
C02388=1022.569,369.743,353.289,172.105,49.188,159.798
C02389=1022.578,369.989,353.249,172.113,49.188,159.799
C02390=1022.586,370.236,353.209,172.121,49.188,159.800
C02391=1022.594,370.482,353.170,172.130,49.188,159.801
C02392=1022.602,370.729,353.129,172.138,49.188,159.803
C02393=1022.612,370.976,353.090,172.146,49.188,159.804
C02394=1022.620,371.222,353.049,172.155,49.188,159.805
C02395=1022.628,371.469,353.010,172.164,49.187,159.806
C02396=1022.636,371.715,352.969,172.172,49.187,159.808
C02397=1022.645,371.962,352.929,172.181,49.187,159.809
C02398=1022.653,372.209,352.889,172.189,49.188,159.810
C02399=1022.662,372.455,352.849,172.197,49.187,159.812
C02400=1022.670,372.702,352.808,172.206,49.187,159.813
C02401=1022.679,372.948,352.768,172.214,49.187,159.814
C02402=1022.687,373.195,352.728,172.224,49.187,159.816
C02403=1022.696,373.442,352.688,172.232,49.187,159.817
C02404=1022.704,373.688,352.647,172.241,49.188,159.818
C02405=1022.713,373.935,352.607,172.249,49.188,159.820
C02406=1022.721,374.181,352.566,172.258,49.188,159.821
C02407=1022.730,374.427,352.526,172.267,49.188,159.823
C02408=1022.739,374.675,352.486,172.275,49.188,159.824
C02409=1022.747,374.921,352.446,172.284,49.188,159.825
C02410=1022.756,375.168,352.405,172.292,49.188,159.827
C02411=1022.765,375.414,352.365,172.302,49.188,159.828
C02412=1022.773,375.661,352.324,172.310,49.188,159.829
C02413=1022.783,375.907,352.284,172.319,49.188,159.831
C02414=1022.791,376.154,352.243,172.328,49.189,159.832
C02415=1022.799,376.401,352.202,172.337,49.189,159.834
C02416=1022.808,376.646,352.162,172.345,49.189,159.835
C02417=1022.817,376.893,352.120,172.354,49.189,159.836
C02418=1022.825,377.139,352.080,172.364,49.189,159.838
C02419=1022.834,377.386,352.039,172.372,49.189,159.839
C02420=1022.843,377.632,351.997,172.381,49.190,159.841
C02421=1022.851,377.879,351.956,172.390,49.190,159.842
C02422=1022.860,378.125,351.916,172.399,49.191,159.844
C02423=1022.869,378.372,351.874,172.408,49.191,159.845
C02424=1022.877,378.618,351.833,172.418,49.191,159.847
C02425=1022.886,378.864,351.792,172.426,49.191,159.848
C02426=1022.895,379.111,351.751,172.435,49.192,159.850
C02427=1022.903,379.357,351.709,172.444,49.192,159.851
C02428=1022.912,379.603,351.668,172.453,49.193,159.853
C02429=1022.921,379.850,351.627,172.462,49.193,159.854
C02430=1022.930,380.096,351.586,172.471,49.193,159.856
C02431=1022.938,380.342,351.544,172.480,49.194,159.857
C02432=1022.947,380.589,351.503,172.490,49.194,159.859
C02433=1022.957,380.847,351.460,172.500,49.195,159.860
C02434=1022.965,381.105,351.416,172.509,49.195,159.862
C02435=1022.975,381.364,351.373,172.519,49.196,159.864
C02436=1022.984,381.622,351.329,172.528,49.196,159.865
C02437=1022.993,381.868,351.288,172.538,49.197,159.867
C02438=1023.003,382.114,351.246,172.547,49.197,159.868
C02439=1023.012,382.360,351.205,172.557,49.198,159.870
C02440=1023.021,382.607,351.163,172.566,49.198,159.872
C02441=1023.030,382.853,351.121,172.575,49.199,159.873
C02442=1023.039,383.100,351.080,172.584,49.200,159.875
C02443=1023.048,383.346,351.038,172.594,49.200,159.876
C02444=1023.056,383.592,350.996,172.603,49.201,159.878
C02445=1023.066,383.838,350.955,172.613,49.201,159.880
C02446=1023.075,384.085,350.913,172.623,49.201,159.881
C02447=1023.084,384.331,350.872,172.631,49.202,159.883
C02448=1023.093,384.577,350.830,172.641,49.202,159.884
C02449=1023.102,384.823,350.787,172.650,49.203,159.886
C02450=1023.111,385.070,350.746,172.660,49.204,159.888
C02451=1023.120,385.316,350.704,172.670,49.204,159.889
C02452=1023.130,385.562,350.661,172.679,49.205,159.891
C02453=1023.140,385.808,350.620,172.689,49.206,159.893
C02454=1023.149,386.055,350.578,172.699,49.207,159.894
C02455=1023.157,386.301,350.535,172.708,49.207,159.896
C02456=1023.166,386.547,350.494,172.718,49.208,159.898
C02457=1023.175,386.793,350.451,172.728,49.209,159.899
C02458=1023.185,387.039,350.408,172.737,49.210,159.901
C02459=1023.194,387.286,350.367,172.747,49.210,159.903
C02460=1023.203,387.531,350.324,172.757,49.211,159.905
C02461=1023.212,387.777,350.282,172.767,49.212,159.906
C02462=1023.221,388.025,350.239,172.776,49.213,159.908
C02463=1023.230,388.270,350.197,172.786,49.214,159.910
C02464=1023.240,388.517,350.154,172.796,49.215,159.912
C02465=1023.250,388.763,350.111,172.806,49.215,159.913
C02466=1023.259,389.008,350.069,172.816,49.216,159.915
C02467=1023.269,389.255,350.026,172.825,49.217,159.917
C02468=1023.277,389.501,349.983,172.836,49.218,159.919
C02469=1023.286,389.747,349.941,172.846,49.219,159.921
C02470=1023.296,389.993,349.898,172.856,49.220,159.922
C02471=1023.305,390.239,349.855,172.866,49.221,159.924
C02472=1023.315,390.485,349.812,172.876,49.221,159.926
C02473=1023.324,390.731,349.770,172.885,49.223,159.928
C02474=1023.334,390.978,349.727,172.896,49.224,159.930
C02475=1023.342,391.223,349.683,172.906,49.225,159.932
C02476=1023.352,391.470,349.640,172.916,49.226,159.933
C02477=1023.362,391.715,349.598,172.926,49.227,159.935
C02478=1023.371,391.961,349.554,172.936,49.228,159.937
C02479=1023.381,392.208,349.511,172.947,49.229,159.939
C02480=1023.390,392.454,349.469,172.957,49.230,159.941
C02481=1023.400,392.699,349.425,172.967,49.231,159.943
C02482=1023.409,392.946,349.382,172.977,49.232,159.945
C02483=1023.419,393.191,349.339,172.988,49.233,159.946
C02484=1023.428,393.438,349.295,172.998,49.235,159.948
C02485=1023.438,393.684,349.252,173.008,49.236,159.950
C02486=1023.447,393.929,349.208,173.019,49.237,159.952
C02487=1023.457,394.176,349.165,173.029,49.238,159.954
C02488=1023.467,394.422,349.122,173.039,49.239,159.956
C02489=1023.476,394.668,349.077,173.050,49.241,159.958
C02490=1023.486,394.913,349.034,173.060,49.242,159.960
C02491=1023.495,395.159,348.990,173.071,49.243,159.962
C02492=1023.505,395.405,348.947,173.081,49.244,159.964
C02493=1023.516,395.700,348.895,173.094,49.246,159.966
C02494=1023.528,395.995,348.842,173.107,49.247,159.969
C02495=1023.540,396.289,348.790,173.120,49.249,159.971
C02496=1023.552,396.585,348.737,173.133,49.250,159.974
C02497=1023.561,396.830,348.693,173.143,49.252,159.976
C02498=1023.571,397.076,348.649,173.154,49.253,159.978
C02499=1023.580,397.322,348.605,173.164,49.255,159.980
C02500=1023.591,397.568,348.562,173.175,49.256,159.982
C02501=1023.600,397.814,348.518,173.186,49.257,159.984
C02502=1023.610,398.060,348.474,173.197,49.258,159.986
C02503=1023.620,398.306,348.429,173.207,49.260,159.988
C02504=1023.631,398.552,348.385,173.218,49.262,159.990
C02505=1023.640,398.798,348.341,173.230,49.263,159.992
C02506=1023.650,399.044,348.297,173.240,49.264,159.994
C02507=1023.660,399.289,348.252,173.251,49.266,159.996
C02508=1023.670,399.535,348.208,173.262,49.267,159.998
C02509=1023.679,399.781,348.163,173.273,49.269,160.001
C02510=1023.690,400.026,348.119,173.284,49.270,160.003
C02511=1023.700,400.273,348.075,173.295,49.272,160.005
C02512=1023.710,400.518,348.030,173.306,49.274,160.007
C02513=1023.720,400.763,347.986,173.318,49.275,160.009
C02514=1023.730,401.009,347.941,173.328,49.276,160.011
C02515=1023.740,401.256,347.896,173.340,49.278,160.014
C02516=1023.749,401.501,347.852,173.351,49.279,160.016
C02517=1023.759,401.747,347.807,173.362,49.281,160.018
C02518=1023.770,401.992,347.763,173.374,49.283,160.020
C02519=1023.780,402.238,347.717,173.384,49.285,160.022
C02520=1023.790,402.484,347.672,173.396,49.286,160.025
C02521=1023.800,402.729,347.627,173.407,49.288,160.027
C02522=1023.810,402.975,347.582,173.419,49.290,160.029
C02523=1023.820,403.220,347.537,173.430,49.291,160.031
C02524=1023.830,403.467,347.492,173.442,49.293,160.034
C02525=1023.840,403.712,347.447,173.454,49.295,160.036
C02526=1023.850,403.958,347.401,173.464,49.297,160.038
C02527=1023.861,404.203,347.357,173.476,49.299,160.040
C02528=1023.871,404.449,347.312,173.487,49.301,160.043
C02529=1023.881,404.694,347.266,173.499,49.302,160.045
C02530=1023.891,404.940,347.221,173.511,49.304,160.047
C02531=1023.902,405.186,347.175,173.522,49.306,160.050
C02532=1023.912,405.431,347.130,173.534,49.308,160.052
C02533=1023.922,405.677,347.084,173.546,49.309,160.054
C02534=1023.933,405.923,347.039,173.558,49.311,160.057
C02535=1023.943,406.168,346.994,173.569,49.314,160.059
C02536=1023.954,406.413,346.948,173.581,49.315,160.061
C02537=1023.964,406.660,346.903,173.593,49.317,160.064
C02538=1023.975,406.905,346.857,173.605,49.319,160.066
C02539=1023.985,407.150,346.812,173.617,49.321,160.069
C02540=1023.996,407.396,346.766,173.628,49.323,160.071
C02541=1024.006,407.641,346.720,173.640,49.325,160.073
C02542=1024.017,407.887,346.674,173.652,49.327,160.076
C02543=1024.027,408.133,346.629,173.665,49.329,160.078
C02544=1024.039,408.378,346.583,173.677,49.331,160.081
C02545=1024.049,408.624,346.537,173.689,49.333,160.083
C02546=1024.060,408.869,346.492,173.701,49.335,160.086
C02547=1024.071,409.114,346.445,173.713,49.337,160.088
C02548=1024.081,409.360,346.399,173.725,49.339,160.091
C02549=1024.092,409.606,346.353,173.738,49.341,160.093
C02550=1024.103,409.851,346.307,173.750,49.343,160.096
C02551=1024.113,410.097,346.260,173.762,49.346,160.098
C02552=1024.123,410.342,346.214,173.775,49.348,160.101
C02553=1024.136,410.634,346.160,173.789,49.350,160.104
C02554=1024.148,410.925,346.104,173.803,49.353,160.107
C02555=1024.162,411.217,346.049,173.818,49.356,160.110
C02556=1024.174,411.508,345.993,173.833,49.358,160.113
C02557=1024.185,411.753,345.947,173.846,49.360,160.116
C02558=1024.196,411.999,345.900,173.858,49.363,160.118
C02559=1024.207,412.244,345.854,173.871,49.365,160.121
C02560=1024.218,412.489,345.807,173.884,49.367,160.124
C02561=1024.229,412.761,345.756,173.898,49.370,160.126
C02562=1024.242,413.032,345.704,173.912,49.373,160.129
C02563=1024.254,413.303,345.652,173.925,49.375,160.132
C02564=1024.267,413.575,345.600,173.939,49.378,160.135
C02565=1024.277,413.820,345.553,173.953,49.380,160.138
C02566=1024.288,414.065,345.506,173.965,49.383,160.141
C02567=1024.300,414.311,345.459,173.978,49.385,160.143
C02568=1024.310,414.556,345.412,173.991,49.387,160.146
C02569=1024.321,414.802,345.365,174.004,49.390,160.149
C02570=1024.333,415.047,345.318,174.017,49.392,160.151
C02571=1024.344,415.292,345.271,174.030,49.394,160.154
C02572=1024.356,415.537,345.224,174.044,49.397,160.157
C02573=1024.366,415.783,345.176,174.056,49.400,160.160
C02574=1024.378,416.028,345.129,174.069,49.402,160.163
C02575=1024.388,416.274,345.081,174.083,49.405,160.165
C02576=1024.400,416.518,345.034,174.095,49.407,160.168
C02577=1024.410,416.764,344.986,174.109,49.410,160.171
C02578=1024.422,417.009,344.938,174.123,49.412,160.174
C02579=1024.433,417.254,344.891,174.136,49.415,160.177
C02580=1024.445,417.499,344.843,174.149,49.418,160.180
C02581=1024.456,417.744,344.796,174.162,49.420,160.183
C02582=1024.467,417.990,344.748,174.176,49.423,160.185
C02583=1024.479,418.235,344.700,174.190,49.426,160.188
C02584=1024.490,418.480,344.652,174.202,49.428,160.191
C02585=1024.501,418.725,344.604,174.217,49.431,160.194
C02586=1024.512,418.970,344.556,174.230,49.434,160.197
C02587=1024.524,419.215,344.508,174.244,49.436,160.200
C02588=1024.535,419.460,344.460,174.257,49.439,160.203
C02589=1024.547,419.705,344.412,174.271,49.442,160.206
C02590=1024.559,419.950,344.363,174.285,49.445,160.209
C02591=1024.570,420.195,344.315,174.299,49.448,160.212
C02592=1024.582,420.441,344.267,174.313,49.450,160.215
C02593=1024.593,420.686,344.219,174.327,49.453,160.218
C02594=1024.605,420.930,344.170,174.341,49.456,160.221
C02595=1024.617,421.176,344.122,174.354,49.459,160.224
C02596=1024.629,421.421,344.073,174.368,49.462,160.227
C02597=1024.641,421.666,344.026,174.382,49.465,160.230
C02598=1024.652,421.911,343.977,174.396,49.468,160.233
C02599=1024.664,422.156,343.929,174.410,49.471,160.236
C02600=1024.676,422.401,343.880,174.426,49.474,160.240
C02601=1024.687,422.646,343.831,174.440,49.476,160.243
C02602=1024.699,422.891,343.782,174.454,49.479,160.246
C02603=1024.711,423.136,343.733,174.468,49.483,160.249
C02604=1024.723,423.381,343.684,174.482,49.486,160.252
C02605=1024.734,423.625,343.635,174.496,49.488,160.255
C02606=1024.747,423.870,343.586,174.511,49.492,160.258
C02607=1024.758,424.115,343.537,174.526,49.495,160.262
C02608=1024.770,424.361,343.488,174.540,49.498,160.265
C02609=1024.782,424.605,343.439,174.555,49.501,160.268
C02610=1024.794,424.851,343.390,174.569,49.504,160.271
C02611=1024.806,425.095,343.341,174.584,49.507,160.275
C02612=1024.818,425.340,343.291,174.599,49.510,160.278
C02613=1024.835,425.669,343.225,174.619,49.515,160.282
C02614=1024.851,425.998,343.159,174.638,49.519,160.287
C02615=1024.867,426.325,343.092,174.658,49.523,160.291
C02616=1024.883,426.653,343.025,174.679,49.528,160.296
C02617=1024.896,426.899,342.976,174.693,49.531,160.299
C02618=1024.908,427.143,342.926,174.709,49.534,160.302
C02619=1024.920,427.387,342.876,174.724,49.537,160.306
C02620=1024.932,427.632,342.826,174.739,49.541,160.309
C02621=1024.944,427.877,342.776,174.754,49.544,160.313
C02622=1024.957,428.122,342.726,174.769,49.548,160.316
C02623=1024.969,428.367,342.676,174.785,49.551,160.320
C02624=1024.981,428.612,342.626,174.800,49.554,160.323
C02625=1024.993,428.856,342.576,174.815,49.558,160.326
C02626=1025.005,429.101,342.526,174.831,49.561,160.330
C02627=1025.018,429.345,342.476,174.846,49.565,160.334
C02628=1025.030,429.590,342.425,174.862,49.568,160.337
C02629=1025.043,429.835,342.375,174.878,49.571,160.341
C02630=1025.055,430.080,342.324,174.893,49.575,160.344
C02631=1025.069,430.324,342.274,174.908,49.579,160.348
C02632=1025.081,430.569,342.224,174.924,49.582,160.351
C02633=1025.094,430.813,342.173,174.940,49.586,160.355
C02634=1025.106,431.058,342.123,174.956,49.590,160.359
C02635=1025.119,431.303,342.072,174.972,49.593,160.362
C02636=1025.132,431.547,342.021,174.988,49.597,160.366
C02637=1025.144,431.792,341.971,175.004,49.600,160.369
C02638=1025.157,432.036,341.920,175.020,49.604,160.373
C02639=1025.170,432.281,341.869,175.037,49.607,160.377
C02640=1025.183,432.525,341.818,175.053,49.611,160.380
C02641=1025.196,432.770,341.767,175.069,49.615,160.384
C02642=1025.208,433.014,341.716,175.085,49.619,160.388
C02643=1025.222,433.259,341.665,175.101,49.622,160.392
C02644=1025.234,433.503,341.614,175.118,49.626,160.395
C02645=1025.248,433.747,341.562,175.134,49.630,160.399
C02646=1025.260,433.992,341.512,175.150,49.634,160.403
C02647=1025.274,434.236,341.460,175.168,49.637,160.407
C02648=1025.287,434.480,341.409,175.184,49.641,160.411
C02649=1025.300,434.725,341.358,175.201,49.645,160.415
C02650=1025.313,434.970,341.305,175.217,49.649,160.418
C02651=1025.325,435.214,341.254,175.234,49.652,160.422
C02652=1025.339,435.458,341.203,175.251,49.656,160.426
C02653=1025.352,435.702,341.151,175.268,49.660,160.430
C02654=1025.365,435.946,341.099,175.285,49.664,160.434
C02655=1025.378,436.191,341.047,175.302,49.668,160.438
C02656=1025.391,436.435,340.995,175.318,49.672,160.442
C02657=1025.405,436.680,340.944,175.336,49.676,160.446
C02658=1025.418,436.924,340.892,175.353,49.680,160.450
C02659=1025.432,437.168,340.839,175.371,49.684,160.454
C02660=1025.445,437.412,340.787,175.387,49.689,160.458
C02661=1025.458,437.656,340.735,175.405,49.692,160.462
C02662=1025.472,437.901,340.683,175.422,49.696,160.466
C02663=1025.485,438.145,340.631,175.440,49.700,160.470
C02664=1025.499,438.389,340.578,175.457,49.704,160.474
C02665=1025.512,438.633,340.526,175.475,49.708,160.478
C02666=1025.526,438.877,340.473,175.493,49.712,160.482
C02667=1025.539,439.121,340.421,175.511,49.717,160.487
C02668=1025.552,439.365,340.368,175.528,49.721,160.491
C02669=1025.567,439.610,340.315,175.546,49.725,160.495
C02670=1025.581,439.853,340.263,175.564,49.730,160.499
C02671=1025.594,440.098,340.210,175.581,49.734,160.503
C02672=1025.607,440.341,340.157,175.600,49.738,160.508
C02673=1025.620,440.553,340.111,175.615,49.741,160.511
C02674=1025.632,440.764,340.066,175.631,49.745,160.515
C02675=1025.644,440.976,340.020,175.647,49.749,160.519
C02676=1025.655,441.187,339.973,175.663,49.753,160.522
C02677=1025.668,441.398,339.927,175.679,49.756,160.526
C02678=1025.680,441.609,339.882,175.695,49.760,160.530
C02679=1025.692,441.820,339.836,175.710,49.764,160.534
C02680=1025.704,442.032,339.790,175.726,49.768,160.537
C02681=1025.718,442.275,339.736,175.746,49.772,160.542
C02682=1025.732,442.518,339.683,175.764,49.777,160.546
C02683=1025.747,442.761,339.631,175.782,49.781,160.551
C02684=1025.762,443.005,339.578,175.801,49.785,160.555
C02685=1025.778,443.248,339.527,175.819,49.789,160.559
C02686=1025.794,443.492,339.475,175.838,49.794,160.564
C02687=1025.810,443.735,339.424,175.857,49.798,160.568
C02688=1025.827,443.979,339.373,175.877,49.801,160.572
C02689=1025.844,444.222,339.323,175.896,49.805,160.577
C02690=1025.862,444.467,339.272,175.915,49.809,160.581
C02691=1025.880,444.711,339.223,175.935,49.813,160.586
C02692=1025.899,444.955,339.174,175.954,49.817,160.590
C02693=1025.918,445.199,339.125,175.973,49.820,160.594
C02694=1025.937,445.443,339.076,175.993,49.823,160.599
C02695=1025.957,445.687,339.028,176.013,49.827,160.603
C02696=1025.978,445.931,338.981,176.033,49.830,160.607
C02697=1025.999,446.176,338.933,176.053,49.834,160.612
C02698=1026.020,446.420,338.887,176.072,49.837,160.616
C02699=1026.042,446.665,338.840,176.092,49.840,160.620
C02700=1026.065,446.910,338.794,176.113,49.843,160.624
C02701=1026.087,447.154,338.748,176.132,49.847,160.629
C02702=1026.110,447.399,338.703,176.153,49.849,160.633
C02703=1026.134,447.644,338.657,176.172,49.852,160.637
C02704=1026.158,447.889,338.613,176.193,49.855,160.642
C02705=1026.183,448.133,338.569,176.214,49.858,160.646
C02706=1026.207,448.378,338.525,176.235,49.861,160.650
C02707=1026.233,448.624,338.482,176.255,49.864,160.655
C02708=1026.258,448.868,338.439,176.276,49.866,160.659
C02709=1026.284,449.113,338.396,176.297,49.869,160.663
C02710=1026.312,449.358,338.354,176.318,49.872,160.668
C02711=1026.340,449.604,338.312,176.339,49.874,160.672
C02712=1026.367,449.849,338.271,176.361,49.876,160.676
C02713=1026.395,450.095,338.230,176.381,49.879,160.680
C02714=1026.423,450.340,338.189,176.402,49.881,160.684
C02715=1026.452,450.585,338.149,176.424,49.883,160.689
C02716=1026.482,450.831,338.109,176.446,49.886,160.693
C02717=1026.512,451.076,338.069,176.468,49.887,160.697
C02718=1026.543,451.322,338.030,176.489,49.889,160.702
C02719=1026.573,451.567,337.991,176.511,49.892,160.706
C02720=1026.605,451.812,337.953,176.533,49.893,160.710
C02721=1026.637,452.059,337.916,176.555,49.895,160.714
C02722=1026.669,452.305,337.877,176.577,49.897,160.719
C02723=1026.702,452.550,337.840,176.600,49.899,160.723
C02724=1026.734,452.795,337.804,176.622,49.901,160.727
C02725=1026.769,453.041,337.768,176.644,49.903,160.732
C02726=1026.803,453.287,337.731,176.667,49.904,160.736
C02727=1026.838,453.533,337.696,176.689,49.906,160.740
C02728=1026.872,453.778,337.660,176.711,49.908,160.744
C02729=1026.908,454.024,337.626,176.735,49.909,160.749
C02730=1026.944,454.271,337.591,176.757,49.910,160.753
C02731=1026.981,454.516,337.558,176.780,49.912,160.757
C02732=1027.017,454.762,337.524,176.803,49.913,160.762
C02733=1026.744,454.840,337.186,176.805,49.972,160.781
C02734=1026.707,454.594,337.219,176.783,49.971,160.777
C02735=1026.671,454.349,337.252,176.760,49.970,160.772
C02736=1026.635,454.103,337.287,176.736,49.968,160.768
C02737=1026.599,453.856,337.322,176.714,49.967,160.764
C02738=1026.564,453.611,337.357,176.691,49.966,160.760
C02739=1026.529,453.366,337.392,176.668,49.964,160.755
C02740=1026.495,453.119,337.428,176.646,49.962,160.751
C02741=1026.461,452.873,337.464,176.624,49.961,160.747
C02742=1026.428,452.628,337.501,176.601,49.959,160.742
C02743=1026.395,452.382,337.537,176.579,49.957,160.738
C02744=1026.363,452.137,337.575,176.556,49.956,160.734
C02745=1026.330,451.890,337.613,176.534,49.954,160.730
C02746=1026.299,451.645,337.651,176.513,49.952,160.725
C02747=1026.268,451.401,337.689,176.490,49.950,160.721
C02748=1026.237,451.154,337.729,176.469,49.948,160.717
C02749=1026.207,450.909,337.768,176.447,49.946,160.713
C02750=1026.177,450.664,337.808,176.425,49.944,160.708
C02751=1026.148,450.418,337.847,176.404,49.942,160.704
C02752=1026.119,450.173,337.888,176.382,49.940,160.700
C02753=1026.091,449.927,337.929,176.361,49.938,160.696
C02754=1026.063,449.682,337.970,176.340,49.935,160.691
C02755=1026.035,449.437,338.012,176.319,49.933,160.687
C02756=1026.009,449.192,338.054,176.298,49.931,160.683
C02757=1025.982,448.947,338.096,176.277,49.928,160.678
C02758=1025.956,448.701,338.140,176.256,49.925,160.674
C02759=1025.930,448.456,338.183,176.235,49.923,160.670
C02760=1025.905,448.211,338.226,176.214,49.921,160.666
C02761=1025.881,447.967,338.271,176.194,49.918,160.661
C02762=1025.856,447.722,338.314,176.173,49.915,160.657
C02763=1025.833,447.477,338.360,176.152,49.912,160.653
C02764=1025.809,447.232,338.405,176.133,49.909,160.648
C02765=1025.786,446.987,338.450,176.112,49.906,160.644
C02766=1025.764,446.743,338.496,176.091,49.903,160.640
C02767=1025.742,446.498,338.543,176.072,49.900,160.636
C02768=1025.721,446.254,338.589,176.052,49.897,160.631
C02769=1025.699,446.009,338.636,176.032,49.894,160.627
C02770=1025.678,445.765,338.683,176.012,49.890,160.622
C02771=1025.658,445.520,338.732,175.992,49.887,160.618
C02772=1025.638,445.276,338.779,175.972,49.884,160.614
C02773=1025.619,445.032,338.828,175.953,49.880,160.610
C02774=1025.600,444.788,338.877,175.933,49.877,160.605
C02775=1025.582,444.544,338.927,175.914,49.874,160.601
C02776=1025.564,444.301,338.976,175.895,49.870,160.597
C02777=1025.546,444.056,339.027,175.876,49.865,160.592
C02778=1025.530,443.812,339.077,175.856,49.862,160.588
C02779=1025.513,443.569,339.128,175.837,49.858,160.584
C02780=1025.496,443.325,339.179,175.818,49.854,160.579
C02781=1025.480,443.082,339.231,175.799,49.850,160.575
C02782=1025.466,442.838,339.283,175.780,49.846,160.570
C02783=1025.450,442.595,339.336,175.762,49.842,160.566
C02784=1025.436,442.352,339.388,175.744,49.838,160.562
C02785=1025.422,442.109,339.442,175.725,49.834,160.557
C02786=1025.410,441.901,339.487,175.709,49.830,160.554
C02787=1025.398,441.694,339.532,175.694,49.827,160.550
C02788=1025.386,441.488,339.577,175.678,49.822,160.546
C02789=1025.374,441.280,339.622,175.662,49.819,160.543
C02790=1025.362,441.073,339.667,175.646,49.815,160.539
C02791=1025.351,440.866,339.713,175.631,49.812,160.535
C02792=1025.339,440.659,339.757,175.615,49.809,160.532
C02793=1025.327,440.452,339.803,175.601,49.805,160.528
C02794=1025.314,440.208,339.855,175.583,49.800,160.524
C02795=1025.300,439.964,339.907,175.564,49.797,160.520
C02796=1025.286,439.721,339.960,175.546,49.792,160.515
C02797=1025.272,439.476,340.014,175.528,49.788,160.511
C02798=1025.259,439.232,340.066,175.511,49.784,160.507
C02799=1025.245,438.988,340.118,175.493,49.780,160.503
C02800=1025.232,438.744,340.171,175.475,49.776,160.499
C02801=1025.218,438.500,340.223,175.458,49.772,160.495
C02802=1025.205,438.256,340.276,175.440,49.768,160.491
C02803=1025.192,438.011,340.328,175.423,49.764,160.486
C02804=1025.178,437.766,340.380,175.405,49.760,160.482
C02805=1025.164,437.523,340.433,175.387,49.756,160.478
C02806=1025.150,437.279,340.485,175.370,49.752,160.474
C02807=1025.137,437.035,340.536,175.352,49.748,160.470
C02808=1025.124,436.791,340.588,175.335,49.745,160.466
C02809=1025.111,436.546,340.641,175.319,49.740,160.462
C02810=1025.097,436.302,340.693,175.301,49.737,160.458
C02811=1025.084,436.058,340.745,175.284,49.733,160.454
C02812=1025.070,435.813,340.797,175.267,49.729,160.450
C02813=1025.058,435.569,340.847,175.250,49.725,160.447
C02814=1025.045,435.324,340.900,175.233,49.722,160.443
C02815=1025.031,435.080,340.952,175.217,49.718,160.439
C02816=1025.018,434.835,341.003,175.200,49.714,160.435
C02817=1025.005,434.592,341.054,175.183,49.710,160.431
C02818=1024.992,434.347,341.106,175.166,49.707,160.427
C02819=1024.979,434.103,341.157,175.150,49.703,160.423
C02820=1024.966,433.858,341.208,175.133,49.699,160.420
C02821=1024.953,433.614,341.259,175.116,49.695,160.416
C02822=1024.941,433.370,341.312,175.100,49.692,160.412
C02823=1024.928,433.125,341.362,175.083,49.688,160.408
C02824=1024.915,432.880,341.414,175.067,49.685,160.405
C02825=1024.902,432.636,341.464,175.051,49.681,160.401
C02826=1024.889,432.391,341.516,175.034,49.678,160.397
C02827=1024.876,432.147,341.566,175.018,49.674,160.393
C02828=1024.863,431.903,341.616,175.002,49.670,160.390
C02829=1024.850,431.658,341.667,174.986,49.667,160.386
C02830=1024.837,431.413,341.718,174.971,49.663,160.383
C02831=1024.825,431.169,341.769,174.955,49.660,160.379
C02832=1024.812,430.924,341.819,174.938,49.657,160.375
C02833=1024.799,430.680,341.870,174.922,49.653,160.372
C02834=1024.787,430.435,341.920,174.906,49.650,160.368
C02835=1024.774,430.191,341.971,174.890,49.646,160.365
C02836=1024.762,429.946,342.021,174.876,49.642,160.361
C02837=1024.749,429.702,342.072,174.860,49.639,160.357
C02838=1024.736,429.457,342.121,174.844,49.636,160.354
C02839=1024.724,429.212,342.171,174.828,49.633,160.350
C02840=1024.712,428.967,342.221,174.813,49.629,160.347
C02841=1024.699,428.723,342.272,174.797,49.626,160.344
C02842=1024.687,428.478,342.322,174.781,49.623,160.340
C02843=1024.674,428.234,342.372,174.767,49.619,160.337
C02844=1024.662,427.989,342.423,174.751,49.616,160.333
C02845=1024.650,427.744,342.473,174.736,49.613,160.330
C02846=1024.638,427.499,342.522,174.721,49.609,160.326
C02847=1024.626,427.254,342.572,174.706,49.607,160.323
C02848=1024.614,427.009,342.622,174.690,49.603,160.319
C02849=1024.601,426.765,342.672,174.675,49.600,160.316
C02850=1024.586,426.434,342.738,174.655,49.595,160.312
C02851=1024.569,426.104,342.806,174.634,49.592,160.307
C02852=1024.552,425.773,342.872,174.614,49.587,160.303
C02853=1024.536,425.441,342.940,174.595,49.583,160.298
C02854=1024.524,425.197,342.989,174.580,49.580,160.295
C02855=1024.512,424.952,343.038,174.565,49.577,160.292
C02856=1024.500,424.707,343.087,174.551,49.574,160.289
C02857=1024.488,424.462,343.136,174.536,49.571,160.285
C02858=1024.476,424.217,343.185,174.521,49.568,160.282
C02859=1024.464,423.973,343.235,174.507,49.565,160.279
C02860=1024.452,423.728,343.283,174.492,49.562,160.276
C02861=1024.440,423.483,343.333,174.478,49.558,160.272
C02862=1024.429,423.238,343.382,174.463,49.556,160.269
C02863=1024.417,422.993,343.430,174.449,49.553,160.266
C02864=1024.405,422.747,343.479,174.434,49.550,160.263
C02865=1024.393,422.503,343.528,174.420,49.547,160.260
C02866=1024.381,422.258,343.576,174.406,49.544,160.257
C02867=1024.369,422.013,343.626,174.392,49.541,160.254
C02868=1024.358,421.767,343.674,174.378,49.538,160.251
C02869=1024.346,421.523,343.722,174.363,49.536,160.247
C02870=1024.335,421.278,343.771,174.349,49.533,160.244
C02871=1024.323,421.033,343.819,174.335,49.530,160.241
C02872=1024.311,420.787,343.868,174.321,49.527,160.238
C02873=1024.299,420.542,343.916,174.307,49.525,160.235
C02874=1024.288,420.297,343.965,174.293,49.522,160.232
C02875=1024.276,420.052,344.012,174.280,49.519,160.229
C02876=1024.265,419.807,344.061,174.266,49.517,160.226
C02877=1024.253,419.562,344.108,174.252,49.514,160.223
C02878=1024.242,419.317,344.157,174.239,49.511,160.220
C02879=1024.230,419.071,344.204,174.224,49.509,160.217
C02880=1024.218,418.826,344.252,174.211,49.506,160.215
C02881=1024.207,418.581,344.300,174.197,49.503,160.211
C02882=1024.195,418.336,344.348,174.184,49.501,160.209
C02883=1024.185,418.091,344.396,174.170,49.498,160.206
C02884=1024.173,417.846,344.444,174.156,49.495,160.203
C02885=1024.162,417.601,344.492,174.143,49.493,160.200
C02886=1024.150,417.356,344.540,174.130,49.490,160.197
C02887=1024.139,417.110,344.587,174.116,49.488,160.194
C02888=1024.128,416.866,344.634,174.103,49.485,160.192
C02889=1024.117,416.620,344.683,174.090,49.483,160.189
C02890=1024.105,416.374,344.730,174.076,49.481,160.186
C02891=1024.095,416.130,344.778,174.063,49.478,160.183
C02892=1024.083,415.884,344.825,174.050,49.476,160.180
C02893=1024.073,415.640,344.873,174.037,49.473,160.177
C02894=1024.061,415.394,344.920,174.023,49.471,160.175
C02895=1024.050,415.148,344.967,174.011,49.468,160.172
C02896=1024.039,414.903,345.013,173.997,49.466,160.169
C02897=1024.028,414.658,345.062,173.985,49.463,160.166
C02898=1024.016,414.412,345.109,173.971,49.462,160.164
C02899=1024.005,414.167,345.155,173.959,49.459,160.161
C02900=1023.994,413.921,345.202,173.946,49.457,160.158
C02901=1023.984,413.676,345.249,173.933,49.454,160.156
C02902=1023.973,413.431,345.296,173.920,49.452,160.153
C02903=1023.961,413.186,345.343,173.908,49.449,160.150
C02904=1023.950,412.941,345.390,173.894,49.448,160.148
C02905=1023.940,412.695,345.435,173.882,49.445,160.145
C02906=1023.929,412.449,345.483,173.870,49.443,160.142
C02907=1023.918,412.204,345.530,173.856,49.441,160.140
C02908=1023.907,411.959,345.576,173.844,49.439,160.137
C02909=1023.896,411.713,345.623,173.831,49.436,160.134
C02910=1023.882,411.394,345.684,173.815,49.434,160.131
C02911=1023.867,411.074,345.744,173.798,49.431,160.128
C02912=1023.854,410.755,345.805,173.782,49.428,160.124
C02913=1023.840,410.434,345.865,173.766,49.425,160.121
C02914=1023.830,410.189,345.911,173.754,49.423,160.118
C02915=1023.819,409.944,345.957,173.741,49.421,160.116
C02916=1023.808,409.699,346.004,173.729,49.419,160.114
C02917=1023.798,409.453,346.050,173.717,49.417,160.111
C02918=1023.787,409.207,346.096,173.705,49.415,160.108
C02919=1023.776,408.962,346.142,173.693,49.413,160.106
C02920=1023.765,408.716,346.188,173.681,49.411,160.103
C02921=1023.755,408.471,346.234,173.669,49.410,160.101
C02922=1023.744,408.225,346.279,173.656,49.407,160.099
C02923=1023.734,407.979,346.325,173.644,49.406,160.096
C02924=1023.723,407.734,346.371,173.632,49.403,160.094
C02925=1023.712,407.488,346.417,173.620,49.402,160.091
C02926=1023.701,407.243,346.462,173.608,49.400,160.089
C02927=1023.691,406.998,346.508,173.596,49.398,160.086
C02928=1023.681,406.752,346.553,173.584,49.396,160.084
C02929=1023.670,406.506,346.599,173.573,49.394,160.082
C02930=1023.659,406.261,346.645,173.561,49.393,160.079
C02931=1023.650,406.015,346.690,173.549,49.390,160.077
C02932=1023.639,405.770,346.736,173.537,49.389,160.075
C02933=1023.628,405.524,346.782,173.525,49.387,160.072
C02934=1023.619,405.278,346.826,173.513,49.385,160.070
C02935=1023.607,405.033,346.872,173.502,49.383,160.068
C02936=1023.597,404.787,346.917,173.490,49.382,160.065
C02937=1023.587,404.541,346.962,173.478,49.380,160.063
C02938=1023.570,404.134,347.038,173.459,49.377,160.059
C02939=1023.553,403.727,347.112,173.441,49.374,160.055
C02940=1023.537,403.320,347.187,173.421,49.372,160.052
C02941=1023.520,402.913,347.261,173.402,49.369,160.048
C02942=1023.509,402.668,347.307,173.390,49.368,160.046
C02943=1023.499,402.422,347.352,173.380,49.366,160.043
C02944=1023.490,402.177,347.396,173.368,49.365,160.041
C02945=1023.479,401.930,347.442,173.357,49.362,160.039
C02946=1023.470,401.685,347.486,173.345,49.361,160.037
C02947=1023.459,401.440,347.531,173.335,49.359,160.035
C02948=1023.450,401.194,347.575,173.323,49.358,160.032
C02949=1023.440,400.947,347.620,173.312,49.356,160.030
C02950=1023.430,400.702,347.665,173.300,49.355,160.028
C02951=1023.419,400.457,347.709,173.290,49.354,160.026
C02952=1023.410,400.211,347.754,173.278,49.352,160.024
C02953=1023.400,399.964,347.798,173.267,49.350,160.022
C02954=1023.389,399.719,347.842,173.256,49.349,160.020
C02955=1023.379,399.474,347.887,173.245,49.348,160.017
C02956=1023.370,399.227,347.931,173.235,49.346,160.015
C02957=1023.360,398.982,347.976,173.223,49.345,160.013
C02958=1023.350,398.736,348.020,173.213,49.344,160.011
C02959=1023.341,398.490,348.064,173.202,49.342,160.009
C02960=1023.330,398.245,348.108,173.190,49.341,160.007
C02961=1023.321,397.999,348.152,173.180,49.340,160.005
C02962=1023.311,397.753,348.196,173.169,49.338,160.003
C02963=1023.301,397.507,348.241,173.158,49.337,160.001
C02964=1023.291,397.261,348.284,173.147,49.336,159.999
C02965=1023.281,397.015,348.328,173.137,49.334,159.997
C02966=1023.266,396.633,348.397,173.120,49.333,159.994
C02967=1023.250,396.252,348.464,173.103,49.330,159.990
C02968=1023.236,395.870,348.532,173.086,49.329,159.987
C02969=1023.221,395.488,348.600,173.071,49.327,159.984
C02970=1023.211,395.243,348.643,173.059,49.326,159.982
C02971=1023.202,394.997,348.687,173.049,49.325,159.980
C02972=1023.192,394.751,348.731,173.038,49.323,159.978
C02973=1023.182,394.505,348.774,173.028,49.322,159.976
C02974=1023.172,394.259,348.818,173.018,49.322,159.975
C02975=1023.163,394.014,348.861,173.007,49.320,159.973
C02976=1023.153,393.767,348.905,172.997,49.319,159.971
C02977=1023.144,393.521,348.948,172.987,49.318,159.969
C02978=1023.135,393.276,348.992,172.975,49.317,159.967
C02979=1023.125,393.029,349.034,172.965,49.316,159.965
C02980=1023.116,392.783,349.078,172.955,49.315,159.963
C02981=1023.106,392.537,349.121,172.945,49.314,159.961
C02982=1023.096,392.291,349.164,172.934,49.313,159.959
C02983=1023.086,392.045,349.207,172.924,49.312,159.957
C02984=1023.078,391.799,349.250,172.914,49.311,159.955
C02985=1023.068,391.553,349.294,172.904,49.310,159.954
C02986=1023.058,391.307,349.336,172.893,49.309,159.952
C02987=1023.049,391.061,349.380,172.883,49.308,159.950
C02988=1023.040,390.815,349.422,172.873,49.307,159.948
C02989=1023.030,390.569,349.465,172.863,49.306,159.946
C02990=1023.021,390.323,349.508,172.853,49.306,159.945
C02991=1023.012,390.076,349.551,172.844,49.305,159.943
C02992=1023.002,389.831,349.594,172.834,49.304,159.941
C02993=1022.992,389.584,349.637,172.823,49.303,159.939
C02994=1022.983,389.339,349.679,172.813,49.302,159.937
C02995=1022.975,389.092,349.722,172.803,49.302,159.936
C02996=1022.965,388.846,349.765,172.793,49.301,159.934
C02997=1022.956,388.600,349.807,172.783,49.300,159.932
C02998=1022.947,388.354,349.849,172.773,49.299,159.930
C02999=1022.937,388.107,349.892,172.764,49.298,159.929
C03000=1022.928,387.861,349.935,172.754,49.297,159.927
C03001=1022.919,387.616,349.977,172.744,49.297,159.925
C03002=1022.910,387.369,350.019,172.734,49.296,159.923
C03003=1022.900,387.123,350.062,172.724,49.296,159.922
C03004=1022.891,386.877,350.104,172.715,49.295,159.920
C03005=1022.882,386.631,350.146,172.705,49.294,159.918
C03006=1022.872,386.384,350.189,172.695,49.294,159.917
C03007=1022.863,386.138,350.230,172.685,49.293,159.915
C03008=1022.854,385.892,350.273,172.676,49.292,159.913
C03009=1022.845,385.646,350.315,172.666,49.292,159.912
C03010=1022.836,385.399,350.356,172.656,49.291,159.910
C03011=1022.827,385.154,350.399,172.646,49.290,159.908
C03012=1022.818,384.907,350.441,172.637,49.290,159.907
C03013=1022.809,384.660,350.482,172.628,49.289,159.905
C03014=1022.800,384.414,350.524,172.618,49.289,159.903
C03015=1022.790,384.168,350.567,172.609,49.288,159.902
C03016=1022.781,383.922,350.608,172.599,49.288,159.900
C03017=1022.772,383.676,350.649,172.589,49.287,159.898
C03018=1022.763,383.429,350.691,172.580,49.287,159.897
C03019=1022.754,383.183,350.733,172.571,49.286,159.895
C03020=1022.745,382.937,350.775,172.561,49.286,159.894
C03021=1022.736,382.690,350.816,172.552,49.285,159.892
C03022=1022.727,382.444,350.858,172.542,49.285,159.890
C03023=1022.718,382.198,350.900,172.534,49.285,159.889
C03024=1022.709,381.952,350.941,172.524,49.284,159.887
C03025=1022.700,381.705,350.983,172.515,49.284,159.886
C03026=1022.691,381.444,351.026,172.505,49.283,159.884
C03027=1022.681,381.184,351.070,172.495,49.283,159.883
C03028=1022.672,380.924,351.114,172.486,49.283,159.881
C03029=1022.662,380.664,351.157,172.476,49.282,159.879
C03030=1022.654,380.418,351.199,172.466,49.282,159.878
C03031=1022.645,380.171,351.240,172.457,49.282,159.876
C03032=1022.636,379.925,351.281,172.448,49.281,159.875
C03033=1022.627,379.678,351.323,172.439,49.281,159.873
C03034=1022.619,379.432,351.364,172.429,49.281,159.872
C03035=1022.609,379.186,351.405,172.421,49.281,159.870
C03036=1022.601,378.939,351.446,172.411,49.280,159.869
C03037=1022.592,378.693,351.488,172.403,49.280,159.867
C03038=1022.584,378.446,351.528,172.394,49.279,159.866
C03039=1022.575,378.200,351.570,172.384,49.280,159.864
C03040=1022.566,377.953,351.611,172.375,49.279,159.863
C03041=1022.558,377.707,351.652,172.366,49.279,159.861
C03042=1022.549,377.461,351.693,172.357,49.279,159.860
C03043=1022.541,377.214,351.733,172.349,49.278,159.858
C03044=1022.532,376.967,351.774,172.339,49.279,159.857
C03045=1022.524,376.722,351.816,172.331,49.278,159.856
C03046=1022.515,376.475,351.857,172.322,49.278,159.854
C03047=1022.506,376.228,351.897,172.312,49.278,159.853
C03048=1022.498,375.982,351.938,172.304,49.278,159.851
C03049=1022.488,375.735,351.978,172.295,49.278,159.850
C03050=1022.480,375.489,352.019,172.286,49.278,159.849
C03051=1022.472,375.242,352.060,172.278,49.278,159.847
C03052=1022.463,374.996,352.100,172.269,49.278,159.846
C03053=1022.454,374.749,352.141,172.260,49.278,159.844
C03054=1022.445,374.503,352.181,172.251,49.278,159.843
C03055=1022.437,374.255,352.221,172.243,49.278,159.842
C03056=1022.428,374.009,352.261,172.233,49.278,159.840
C03057=1022.420,373.762,352.302,172.225,49.278,159.839
C03058=1022.411,373.516,352.342,172.217,49.278,159.838
C03059=1022.403,373.269,352.382,172.208,49.278,159.836
C03060=1022.394,373.023,352.423,172.199,49.278,159.835
C03061=1022.386,372.776,352.463,172.190,49.278,159.834
C03062=1022.377,372.530,352.503,172.182,49.278,159.832
C03063=1022.369,372.283,352.544,172.174,49.278,159.831
C03064=1022.360,372.037,352.584,172.165,49.278,159.830
C03065=1022.352,371.790,352.623,172.156,49.278,159.828
C03066=1022.343,371.543,352.664,172.148,49.279,159.827
C03067=1022.335,371.296,352.704,172.139,49.279,159.826
C03068=1022.326,371.050,352.744,172.131,49.279,159.825
C03069=1022.319,370.803,352.784,172.123,49.279,159.823
C03070=1022.310,370.557,352.824,172.114,49.279,159.822
C03071=1022.302,370.310,352.864,172.105,49.280,159.821
C03072=1022.293,370.063,352.903,172.097,49.280,159.819
C03073=1022.285,369.817,352.944,172.089,49.280,159.818
C03074=1022.277,369.570,352.983,172.080,49.280,159.817
C03075=1022.269,369.323,353.023,172.072,49.280,159.816
C03076=1022.260,369.078,353.063,172.063,49.280,159.814
C03077=1022.252,368.831,353.103,172.055,49.281,159.813
C03078=1022.243,368.583,353.143,172.047,49.281,159.812
C03079=1022.236,368.336,353.183,172.039,49.281,159.811
C03080=1022.227,368.090,353.222,172.031,49.281,159.810
C03081=1022.219,367.843,353.261,172.022,49.282,159.808
C03082=1022.211,367.601,353.300,172.014,49.282,159.807
C03083=1022.202,367.359,353.339,172.006,49.282,159.806
C03084=1022.194,367.116,353.378,171.998,49.283,159.805
C03085=1022.186,366.874,353.417,171.990,49.283,159.804
C03086=1022.178,366.631,353.456,171.982,49.284,159.803
C03087=1022.169,366.389,353.494,171.974,49.284,159.801
C03088=1022.162,366.145,353.532,171.965,49.285,159.800
C03089=1022.154,365.903,353.571,171.957,49.285,159.799
C03090=1022.146,365.657,353.610,171.949,49.285,159.798
C03091=1022.137,365.410,353.650,171.941,49.286,159.797
C03092=1022.129,365.163,353.689,171.933,49.286,159.796
C03093=1022.121,364.916,353.728,171.925,49.287,159.794
C03094=1022.112,364.670,353.767,171.917,49.287,159.793
C03095=1022.105,364.423,353.807,171.909,49.288,159.792
C03096=1022.097,364.176,353.845,171.901,49.288,159.791
C03097=1022.089,363.930,353.884,171.893,49.289,159.790
C03098=1022.080,363.682,353.923,171.885,49.290,159.789
C03099=1022.072,363.436,353.962,171.877,49.290,159.788
C03100=1022.064,363.189,354.001,171.869,49.291,159.787
C03101=1022.055,362.942,354.040,171.861,49.291,159.785
C03102=1022.048,362.695,354.079,171.853,49.292,159.785
C03103=1022.040,362.449,354.119,171.845,49.293,159.783
C03104=1022.032,362.201,354.157,171.838,49.293,159.782
C03105=1022.024,361.954,354.196,171.829,49.293,159.781
C03106=1022.016,361.708,354.235,171.822,49.294,159.780
C03107=1022.008,361.461,354.273,171.814,49.295,159.779
C03108=1022.000,361.213,354.312,171.805,49.295,159.778
C03109=1021.992,360.968,354.351,171.798,49.296,159.777
C03110=1021.984,360.720,354.390,171.790,49.297,159.776
C03111=1021.976,360.473,354.429,171.783,49.297,159.775
C03112=1021.969,360.227,354.467,171.775,49.298,159.774
C03113=1021.960,359.980,354.506,171.767,49.299,159.773
C03114=1021.953,359.734,354.544,171.759,49.299,159.772
C03115=1021.944,359.486,354.583,171.751,49.300,159.771
C03116=1021.936,359.239,354.622,171.743,49.301,159.770
C03117=1021.929,358.993,354.660,171.735,49.302,159.769
C03118=1021.921,358.745,354.699,171.729,49.303,159.768
C03119=1021.913,358.499,354.737,171.720,49.303,159.767
C03120=1021.905,358.251,354.775,171.713,49.304,159.766
C03121=1021.898,358.005,354.813,171.705,49.305,159.765
C03122=1021.890,357.757,354.852,171.697,49.306,159.764
C03123=1021.881,357.511,354.889,171.690,49.306,159.763
C03124=1021.873,357.264,354.928,171.682,49.307,159.762
C03125=1021.866,357.017,354.965,171.675,49.308,159.761
C03126=1021.858,356.770,355.004,171.667,49.309,159.760
C03127=1021.850,356.523,355.042,171.659,49.310,159.759
C03128=1021.842,356.276,355.081,171.652,49.311,159.758
C03129=1021.834,356.029,355.118,171.644,49.312,159.757
C03130=1021.826,355.782,355.156,171.637,49.313,159.756
C03131=1021.818,355.535,355.195,171.629,49.314,159.755
C03132=1021.810,355.287,355.232,171.622,49.315,159.754
C03133=1021.803,355.041,355.271,171.614,49.316,159.753
C03134=1021.796,354.794,355.308,171.607,49.317,159.752
C03135=1021.787,354.547,355.346,171.599,49.318,159.751
C03136=1021.780,354.300,355.384,171.592,49.318,159.750
C03137=1021.772,354.053,355.422,171.584,49.319,159.749
C03138=1021.764,353.805,355.460,171.577,49.321,159.748
C03139=1021.756,353.559,355.497,171.570,49.321,159.748
C03140=1021.749,353.312,355.535,171.562,49.322,159.747
C03141=1021.740,353.064,355.572,171.555,49.324,159.746
C03142=1021.734,352.826,355.608,171.548,49.325,159.745
C03143=1021.726,352.587,355.646,171.540,49.326,159.744
C03144=1021.718,352.348,355.681,171.534,49.326,159.743
C03145=1021.711,352.109,355.718,171.526,49.328,159.742
C03146=1021.703,351.870,355.754,171.519,49.329,159.742
C03147=1021.696,351.631,355.791,171.512,49.330,159.741
C03148=1021.688,351.392,355.826,171.505,49.331,159.740
C03149=1021.681,351.152,355.863,171.498,49.332,159.739
C03150=1021.674,350.905,355.900,171.491,49.334,159.738
C03151=1021.666,350.658,355.937,171.483,49.335,159.737
C03152=1021.659,350.411,355.975,171.477,49.335,159.736
C03153=1021.650,350.164,356.012,171.469,49.337,159.736
C03154=1021.643,349.916,356.050,171.461,49.338,159.735
C03155=1021.635,349.669,356.087,171.455,49.339,159.734
C03156=1021.627,349.422,356.124,171.447,49.341,159.733
C03157=1021.620,349.175,356.162,171.440,49.342,159.732
C03158=1021.613,348.928,356.199,171.433,49.343,159.731
C03159=1021.605,348.681,356.236,171.425,49.344,159.731
C03160=1021.598,348.434,356.274,171.419,49.345,159.730
C03161=1021.590,348.187,356.311,171.412,49.347,159.729
C03162=1021.583,347.940,356.348,171.404,49.348,159.728
C03163=1021.575,347.693,356.384,171.398,49.349,159.727
C03164=1021.568,347.446,356.422,171.390,49.350,159.727
C03165=1021.560,347.199,356.459,171.383,49.352,159.726
C03166=1021.553,346.951,356.496,171.376,49.353,159.725
C03167=1021.545,346.704,356.533,171.370,49.355,159.724
C03168=1021.537,346.457,356.569,171.362,49.356,159.723
C03169=1021.530,346.210,356.606,171.355,49.357,159.723
C03170=1021.522,345.963,356.643,171.348,49.359,159.722
C03171=1021.515,345.715,356.680,171.341,49.360,159.721
C03172=1021.507,345.468,356.717,171.334,49.362,159.721
C03173=1021.499,345.221,356.753,171.327,49.363,159.720
C03174=1021.492,344.974,356.791,171.320,49.364,159.719
C03175=1021.485,344.727,356.827,171.313,49.366,159.718
C03176=1021.477,344.480,356.863,171.306,49.367,159.718
C03177=1021.470,344.232,356.900,171.299,49.369,159.717
C03178=1021.462,343.985,356.937,171.293,49.370,159.716
C03179=1021.454,343.738,356.973,171.285,49.372,159.715
C03180=1021.447,343.490,357.010,171.279,49.373,159.715
C03181=1021.440,343.244,357.046,171.272,49.375,159.714
C03182=1021.432,342.997,357.083,171.265,49.376,159.713
C03183=1021.425,342.749,357.120,171.258,49.378,159.712
C03184=1021.418,342.502,357.156,171.251,49.379,159.712
C03185=1021.410,342.254,357.192,171.244,49.381,159.711
C03186=1021.404,342.007,357.229,171.238,49.382,159.710
C03187=1021.396,341.760,357.266,171.230,49.384,159.710
C03188=1021.388,341.513,357.302,171.224,49.385,159.709
C03189=1021.381,341.266,357.338,171.217,49.388,159.708
C03190=1021.374,341.018,357.375,171.210,49.389,159.708
C03191=1021.366,340.771,357.411,171.203,49.391,159.707
C03192=1021.359,340.523,357.447,171.197,49.392,159.706
C03193=1021.352,340.277,357.483,171.189,49.394,159.706
C03194=1021.345,340.029,357.520,171.183,49.395,159.705
C03195=1021.338,339.782,357.555,171.176,49.397,159.704
C03196=1021.330,339.535,357.592,171.169,49.398,159.704
C03197=1021.322,339.287,357.628,171.163,49.400,159.703
C03198=1021.315,339.041,357.664,171.156,49.402,159.702
C03199=1021.308,338.792,357.699,171.150,49.403,159.702
C03200=1021.300,338.545,357.735,171.143,49.406,159.701
C03201=1021.293,338.298,357.771,171.136,49.407,159.700
C03202=1021.287,338.058,357.806,171.129,49.409,159.700
C03203=1021.279,337.817,357.841,171.123,49.411,159.699
C03204=1021.272,337.577,357.877,171.117,49.413,159.699
C03205=1021.265,337.336,357.911,171.110,49.414,159.698
C03206=1021.258,337.095,357.946,171.103,49.416,159.698
C03207=1021.250,336.854,357.981,171.097,49.418,159.697
C03208=1021.243,336.614,358.015,171.091,49.420,159.696
C03209=1021.237,336.373,358.050,171.085,49.421,159.696
C03210=1021.229,336.126,358.086,171.078,49.423,159.695
C03211=1021.222,335.879,358.122,171.071,49.425,159.694
C03212=1021.215,335.631,358.158,171.065,49.427,159.694
C03213=1021.208,335.384,358.193,171.058,49.429,159.693
C03214=1021.201,335.137,358.229,171.052,49.430,159.693
C03215=1021.193,334.889,358.264,171.045,49.432,159.692
C03216=1021.186,334.642,358.300,171.039,49.434,159.692
C03217=1021.179,334.394,358.336,171.032,49.436,159.691
C03218=1021.172,334.147,358.371,171.025,49.438,159.690
C03219=1021.165,333.900,358.407,171.019,49.440,159.690
C03220=1021.158,333.652,358.442,171.013,49.442,159.689
C03221=1021.151,333.405,358.478,171.006,49.444,159.689
C03222=1021.144,333.158,358.513,171.000,49.446,159.688
C03223=1021.137,332.910,358.549,170.994,49.448,159.688
C03224=1021.129,332.663,358.584,170.987,49.450,159.687
C03225=1021.122,332.416,358.619,170.981,49.452,159.687
C03226=1021.115,332.168,358.654,170.974,49.454,159.686
C03227=1021.108,331.921,358.690,170.968,49.456,159.686
C03228=1021.101,331.673,358.725,170.961,49.457,159.685
C03229=1021.093,331.425,358.760,170.954,49.460,159.684
C03230=1021.086,331.178,358.795,170.948,49.462,159.684
C03231=1021.079,330.931,358.831,170.942,49.464,159.683
C03232=1021.072,330.684,358.866,170.935,49.466,159.683
C03233=1021.064,330.436,358.901,170.929,49.468,159.682
C03234=1021.057,330.189,358.936,170.923,49.471,159.682
C03235=1021.051,329.942,358.971,170.916,49.473,159.682
C03236=1021.044,329.694,359.006,170.910,49.475,159.681
C03237=1021.036,329.446,359.040,170.904,49.477,159.681
C03238=1021.029,329.198,359.075,170.897,49.479,159.680
C03239=1021.023,328.951,359.111,170.891,49.481,159.680
C03240=1021.015,328.704,359.145,170.885,49.483,159.679
C03241=1021.008,328.457,359.180,170.878,49.485,159.678
C03242=1021.002,328.209,359.215,170.872,49.487,159.678
C03243=1020.995,327.962,359.250,170.867,49.490,159.678
C03244=1020.987,327.715,359.285,170.861,49.492,159.677
C03245=1020.980,327.466,359.320,170.853,49.494,159.677
C03246=1020.973,327.219,359.355,170.847,49.496,159.676
C03247=1020.967,326.971,359.390,170.842,49.499,159.676
C03248=1020.959,326.724,359.425,170.835,49.501,159.675
C03249=1020.953,326.476,359.459,170.829,49.503,159.675
C03250=1020.945,326.229,359.494,170.823,49.506,159.675
C03251=1020.938,325.982,359.527,170.816,49.508,159.674
C03252=1020.931,325.734,359.563,170.810,49.510,159.674
C03253=1020.924,325.487,359.596,170.804,49.512,159.673
C03254=1020.916,325.240,359.631,170.797,49.515,159.673
C03255=1020.909,324.992,359.665,170.792,49.517,159.672
C03256=1020.903,324.745,359.700,170.786,49.520,159.672
C03257=1020.895,324.497,359.734,170.779,49.522,159.672
C03258=1020.888,324.249,359.768,170.773,49.525,159.671
C03259=1020.881,324.002,359.803,170.767,49.527,159.671
C03260=1020.874,323.754,359.836,170.762,49.529,159.670
C03261=1020.867,323.506,359.870,170.755,49.532,159.670
C03262=1020.860,323.263,359.905,170.749,49.534,159.670
C03263=1020.853,323.021,359.938,170.743,49.537,159.669
C03264=1020.846,322.778,359.972,170.737,49.539,159.669
C03265=1020.839,322.535,360.004,170.732,49.542,159.669
C03266=1020.832,322.292,360.039,170.725,49.544,159.668
C03267=1020.825,322.050,360.072,170.719,49.546,159.668
C03268=1020.819,321.807,360.106,170.713,49.549,159.667
C03269=1020.812,321.564,360.138,170.708,49.552,159.667
C03270=1020.804,321.316,360.172,170.701,49.554,159.667
C03271=1020.798,321.069,360.207,170.695,49.557,159.666
C03272=1020.791,320.821,360.241,170.689,49.559,159.666
C03273=1020.783,320.574,360.275,170.684,49.562,159.666
C03274=1020.777,320.326,360.309,170.677,49.564,159.665
C03275=1020.770,320.079,360.343,170.671,49.567,159.665
C03276=1020.763,319.831,360.377,170.665,49.569,159.665
C03277=1020.756,319.583,360.411,170.659,49.572,159.664
C03278=1020.749,319.335,360.445,170.654,49.575,159.664
C03279=1020.743,319.088,360.479,170.647,49.577,159.664
C03280=1020.736,318.841,360.512,170.641,49.579,159.663
C03281=1020.728,318.593,360.546,170.635,49.582,159.663
C03282=1020.722,318.345,360.581,170.630,49.585,159.662
C03283=1020.715,318.098,360.614,170.624,49.587,159.662
C03284=1020.708,317.850,360.648,170.617,49.590,159.662
C03285=1020.702,317.602,360.682,170.612,49.593,159.662
C03286=1020.695,317.355,360.716,170.606,49.595,159.661
C03287=1020.688,317.108,360.750,170.600,49.598,159.661
C03288=1020.681,316.859,360.783,170.595,49.601,159.661
C03289=1020.675,316.612,360.817,170.588,49.604,159.660
C03290=1020.668,316.365,360.851,170.582,49.606,159.660
C03291=1020.661,316.117,360.884,170.577,49.609,159.660
C03292=1020.654,315.870,360.918,170.571,49.611,159.659
C03293=1020.648,315.622,360.952,170.565,49.614,159.659
C03294=1020.641,315.374,360.985,170.559,49.617,159.659
C03295=1020.634,315.127,361.019,170.553,49.620,159.658
C03296=1020.628,314.880,361.052,170.547,49.622,159.658
C03297=1020.621,314.631,361.086,170.542,49.626,159.658
C03298=1020.614,314.383,361.120,170.537,49.628,159.658
C03299=1020.608,314.136,361.153,170.531,49.631,159.657
C03300=1020.600,313.889,361.187,170.524,49.634,159.657
C03301=1020.595,313.641,361.220,170.519,49.636,159.657
C03302=1020.588,313.393,361.254,170.513,49.639,159.657
C03303=1020.581,313.146,361.287,170.507,49.642,159.656
C03304=1020.574,312.898,361.321,170.502,49.645,159.656
C03305=1020.568,312.651,361.355,170.496,49.647,159.656
C03306=1020.562,312.403,361.388,170.491,49.650,159.656
C03307=1020.555,312.155,361.421,170.484,49.653,159.655
C03308=1020.549,311.908,361.454,170.479,49.656,159.655
C03309=1020.541,311.660,361.488,170.473,49.659,159.655
C03310=1020.536,311.412,361.521,170.467,49.661,159.654
C03311=1020.529,311.165,361.555,170.462,49.665,159.654
C03312=1020.522,310.917,361.588,170.456,49.667,159.654
C03313=1020.516,310.670,361.621,170.451,49.670,159.654
C03314=1020.510,310.421,361.655,170.445,49.673,159.654
C03315=1020.503,310.174,361.689,170.440,49.676,159.653
C03316=1020.497,309.927,361.721,170.433,49.679,159.653
C03317=1020.489,309.679,361.754,170.428,49.682,159.653
C03318=1020.483,309.431,361.787,170.422,49.685,159.653
C03319=1020.476,309.184,361.819,170.417,49.688,159.653
C03320=1020.469,308.936,361.852,170.411,49.691,159.652
C03321=1020.462,308.688,361.885,170.405,49.695,159.652
C03322=1020.456,308.447,361.917,170.399,49.697,159.652
C03323=1020.450,308.208,361.948,170.394,49.701,159.652
C03324=1020.442,307.967,361.980,170.389,49.703,159.652
C03325=1020.436,307.727,362.011,170.383,49.707,159.651
C03326=1020.429,307.487,362.043,170.378,49.710,159.651
C03327=1020.423,307.247,362.075,170.372,49.712,159.651
C03328=1020.416,307.006,362.107,170.367,49.716,159.651
C03329=1020.409,306.767,362.138,170.362,49.719,159.651
C03330=1020.403,306.519,362.171,170.356,49.722,159.651
C03331=1020.397,306.270,362.203,170.351,49.725,159.650
C03332=1020.390,306.023,362.235,170.345,49.728,159.650
C03333=1020.383,305.775,362.268,170.339,49.732,159.650
C03334=1020.376,305.528,362.300,170.334,49.735,159.650
C03335=1020.369,305.280,362.333,170.329,49.738,159.650
C03336=1020.363,305.032,362.366,170.323,49.742,159.650
C03337=1020.355,304.784,362.398,170.318,49.744,159.650
C03338=1020.349,304.536,362.430,170.312,49.747,159.649
C03339=1020.342,304.289,362.462,170.306,49.751,159.649
C03340=1020.336,304.041,362.495,170.301,49.754,159.649
C03341=1020.329,303.794,362.527,170.295,49.758,159.649
C03342=1020.322,303.545,362.560,170.290,49.761,159.649
C03343=1020.316,303.297,362.592,170.285,49.764,159.649
C03344=1020.309,303.050,362.625,170.279,49.767,159.649
C03345=1020.303,302.802,362.657,170.274,49.771,159.649
C03346=1020.296,302.555,362.689,170.268,49.774,159.649
C03347=1020.290,302.307,362.722,170.263,49.778,159.648
C03348=1020.284,302.059,362.754,170.257,49.781,159.648
C03349=1020.277,301.812,362.786,170.252,49.784,159.648
C03350=1020.270,301.563,362.818,170.247,49.787,159.648
C03351=1020.263,301.315,362.850,170.241,49.791,159.648
C03352=1020.257,301.068,362.883,170.236,49.794,159.648
C03353=1020.251,300.820,362.915,170.230,49.798,159.648
C03354=1020.244,300.572,362.947,170.225,49.801,159.648
C03355=1020.238,300.324,362.979,170.219,49.804,159.648
C03356=1020.231,300.077,363.011,170.214,49.807,159.647
C03357=1020.225,299.829,363.043,170.209,49.811,159.648
C03358=1020.218,299.581,363.076,170.204,49.815,159.647
C03359=1020.212,299.333,363.108,170.198,49.818,159.647
C03360=1020.206,299.086,363.140,170.193,49.821,159.647
C03361=1020.199,298.838,363.172,170.188,49.825,159.647
C03362=1020.193,298.589,363.204,170.182,49.828,159.647
C03363=1020.186,298.342,363.236,170.177,49.832,159.647
C03364=1020.180,298.094,363.268,170.171,49.835,159.647
C03365=1020.174,297.846,363.300,170.166,49.839,159.647
C03366=1020.167,297.598,363.332,170.161,49.842,159.647
C03367=1020.161,297.350,363.364,170.155,49.845,159.647
C03368=1020.154,297.102,363.396,170.151,49.849,159.647
C03369=1020.148,296.855,363.428,170.145,49.852,159.647
C03370=1020.141,296.607,363.460,170.140,49.856,159.646
C03371=1020.136,296.359,363.491,170.135,49.860,159.647
C03372=1020.129,296.112,363.524,170.130,49.863,159.646
C03373=1020.123,295.864,363.556,170.123,49.867,159.646
C03374=1020.117,295.616,363.588,170.118,49.870,159.646
C03375=1020.110,295.368,363.619,170.113,49.874,159.646
C03376=1020.104,295.119,363.651,170.108,49.877,159.646
C03377=1020.097,294.872,363.683,170.103,49.881,159.646
C03378=1020.092,294.625,363.715,170.098,49.884,159.646
C03379=1020.086,294.376,363.747,170.092,49.888,159.646
C03380=1020.079,294.129,363.778,170.087,49.891,159.646
C03381=1020.073,293.880,363.810,170.082,49.895,159.646
C03382=1020.067,293.649,363.840,170.077,49.899,159.646
C03383=1020.061,293.418,363.870,170.073,49.902,159.646
C03384=1020.055,293.186,363.899,170.068,49.905,159.646
C03385=1020.049,292.955,363.928,170.063,49.909,159.646
C03386=1020.043,292.724,363.958,170.057,49.912,159.646
C03387=1020.037,292.492,363.987,170.053,49.915,159.646
C03388=1020.031,292.260,364.017,170.048,49.919,159.646
C03389=1020.025,292.029,364.045,170.043,49.922,159.646
C03390=1020.019,291.781,364.077,170.038,49.926,159.646
C03391=1020.013,291.533,364.109,170.033,49.930,159.646
C03392=1020.006,291.285,364.140,170.028,49.934,159.646
C03393=1019.999,291.037,364.171,170.023,49.938,159.646
C03394=1019.993,290.790,364.202,170.018,49.941,159.646
C03395=1019.987,290.542,364.233,170.013,49.945,159.646
C03396=1019.980,290.294,364.265,170.007,49.949,159.646
C03397=1019.974,290.045,364.295,170.002,49.953,159.646
C03398=1019.968,289.798,364.327,169.997,49.957,159.646
C03399=1019.961,289.550,364.358,169.992,49.961,159.646
C03400=1019.955,289.301,364.389,169.987,49.965,159.646
C03401=1019.948,289.053,364.421,169.982,49.968,159.646
C03402=1019.942,288.806,364.452,169.977,49.972,159.646
C03403=1019.936,288.558,364.482,169.972,49.976,159.646
C03404=1019.929,288.310,364.514,169.966,49.980,159.646
C03405=1019.923,288.062,364.544,169.961,49.984,159.647
C03406=1019.916,287.814,364.576,169.956,49.988,159.647
C03407=1019.910,287.566,364.607,169.951,49.992,159.647
C03408=1019.904,287.318,364.637,169.946,49.996,159.647
C03409=1019.897,287.070,364.669,169.941,50.000,159.647
C03410=1019.891,286.823,364.699,169.937,50.004,159.647
C03411=1019.885,286.574,364.730,169.932,50.008,159.647
C03412=1019.878,286.326,364.761,169.927,50.012,159.647
C03413=1019.872,286.078,364.792,169.921,50.016,159.647
C03414=1019.866,285.830,364.823,169.916,50.020,159.647
C03415=1019.859,285.582,364.854,169.911,50.024,159.647
C03416=1019.853,285.335,364.885,169.906,50.028,159.647
C03417=1019.847,285.086,364.916,169.901,50.032,159.648
C03418=1019.841,284.838,364.946,169.896,50.036,159.648
C03419=1019.834,284.590,364.977,169.891,50.040,159.648
C03420=1019.828,284.343,365.008,169.886,50.044,159.648
C03421=1019.822,284.094,365.038,169.880,50.048,159.648
C03422=1019.815,283.847,365.068,169.876,50.052,159.648
C03423=1019.809,283.598,365.099,169.871,50.057,159.648
C03424=1019.802,283.350,365.130,169.866,50.061,159.648
C03425=1019.796,283.102,365.161,169.861,50.065,159.648
C03426=1019.789,282.854,365.191,169.856,50.069,159.648
C03427=1019.783,282.606,365.221,169.851,50.074,159.649
C03428=1019.777,282.358,365.252,169.846,50.078,159.649
C03429=1019.771,282.110,365.282,169.841,50.082,159.649
C03430=1019.765,281.861,365.313,169.836,50.086,159.649
C03431=1019.758,281.614,365.343,169.831,50.090,159.649
C03432=1019.752,281.366,365.374,169.827,50.094,159.649
C03433=1019.746,281.118,365.405,169.822,50.098,159.649
C03434=1019.739,280.870,365.435,169.817,50.103,159.650
C03435=1019.733,280.622,365.465,169.811,50.107,159.650
C03436=1019.727,280.374,365.495,169.806,50.111,159.650
C03437=1019.721,280.126,365.526,169.802,50.116,159.650
C03438=1019.715,279.878,365.556,169.797,50.120,159.650
C03439=1019.708,279.629,365.587,169.792,50.124,159.650
C03440=1019.702,279.382,365.617,169.787,50.128,159.650
C03441=1019.696,279.134,365.647,169.782,50.132,159.651
C03442=1019.690,278.909,365.675,169.778,50.136,159.651
C03443=1019.685,278.683,365.703,169.773,50.140,159.651
C03444=1019.679,278.458,365.730,169.769,50.144,159.651
C03445=1019.673,278.232,365.758,169.764,50.148,159.651
C03446=1019.668,278.007,365.785,169.760,50.152,159.651
C03447=1019.662,277.781,365.812,169.755,50.156,159.651
C03448=1019.657,277.556,365.840,169.752,50.160,159.652
C03449=1019.651,277.330,365.867,169.747,50.164,159.652
C03450=1019.645,277.083,365.897,169.742,50.168,159.652
C03451=1019.638,276.834,365.927,169.737,50.172,159.652
C03452=1019.632,276.587,365.958,169.733,50.177,159.652
C03453=1019.627,276.339,365.988,169.728,50.182,159.653
C03454=1019.620,276.090,366.017,169.722,50.186,159.653
C03455=1019.614,275.842,366.048,169.718,50.191,159.653
C03456=1019.607,275.595,366.077,169.713,50.195,159.653
C03457=1019.601,275.346,366.107,169.708,50.199,159.653
C03458=1019.595,275.098,366.137,169.704,50.204,159.654
C03459=1019.589,274.850,366.167,169.699,50.208,159.654
C03460=1019.582,274.601,366.197,169.693,50.213,159.654
C03461=1019.576,274.354,366.227,169.689,50.217,159.654
C03462=1019.570,274.105,366.256,169.684,50.222,159.654
C03463=1019.564,273.858,366.287,169.680,50.227,159.655
C03464=1019.557,273.609,366.316,169.675,50.231,159.655
C03465=1019.552,273.361,366.346,169.670,50.235,159.655
C03466=1019.545,273.113,366.375,169.666,50.240,159.655
C03467=1019.539,272.865,366.406,169.660,50.245,159.655
C03468=1019.533,272.616,366.435,169.655,50.249,159.656
C03469=1019.527,272.368,366.466,169.651,50.254,159.656
C03470=1019.521,272.120,366.495,169.646,50.258,159.656
C03471=1019.515,271.872,366.525,169.642,50.263,159.656
C03472=1019.508,271.624,366.554,169.637,50.268,159.657
C03473=1019.502,271.375,366.583,169.632,50.273,159.657
C03474=1019.496,271.128,366.614,169.627,50.277,159.657
C03475=1019.490,270.879,366.643,169.623,50.282,159.657
C03476=1019.484,270.632,366.673,169.618,50.286,159.657
C03477=1019.477,270.383,366.702,169.613,50.290,159.658
C03478=1019.472,270.135,366.732,169.609,50.295,159.658
C03479=1019.465,269.886,366.761,169.603,50.300,159.658
C03480=1019.459,269.639,366.791,169.599,50.305,159.659
C03481=1019.453,269.390,366.821,169.594,50.309,159.659
C03482=1019.447,269.142,366.850,169.590,50.314,159.659
C03483=1019.440,268.895,366.879,169.585,50.319,159.659
C03484=1019.435,268.646,366.909,169.580,50.324,159.660
C03485=1019.428,268.398,366.938,169.575,50.329,159.660
C03486=1019.422,268.150,366.967,169.571,50.334,159.660
C03487=1019.416,267.902,366.996,169.566,50.338,159.661
C03488=1019.410,267.653,367.026,169.562,50.343,159.661
C03489=1019.404,267.404,367.055,169.557,50.348,159.661
C03490=1019.397,267.157,367.085,169.552,50.353,159.661
C03491=1019.391,266.909,367.114,169.547,50.357,159.662
C03492=1019.385,266.660,367.144,169.543,50.362,159.662
C03493=1019.379,266.412,367.173,169.539,50.367,159.662
C03494=1019.373,266.164,367.202,169.534,50.372,159.663
C03495=1019.367,265.916,367.231,169.529,50.377,159.663
C03496=1019.360,265.668,367.260,169.524,50.382,159.663
C03497=1019.355,265.419,367.289,169.520,50.386,159.663
C03498=1019.349,265.171,367.318,169.515,50.392,159.664
C03499=1019.342,264.923,367.347,169.511,50.396,159.664
C03500=1019.336,264.675,367.377,169.505,50.401,159.664
C03501=1019.330,264.427,367.406,169.501,50.407,159.665
C03502=1019.324,264.203,367.432,169.497,50.411,159.665
C03503=1019.319,263.980,367.457,169.493,50.415,159.665
C03504=1019.314,263.757,367.484,169.488,50.420,159.665
C03505=1019.308,263.535,367.509,169.485,50.424,159.666
C03506=1019.302,263.311,367.535,169.480,50.429,159.666
C03507=1019.297,263.088,367.562,169.477,50.433,159.667
C03508=1019.292,262.865,367.587,169.472,50.438,159.667
C03509=1019.286,262.642,367.613,169.468,50.442,159.667
C03510=1019.280,262.394,367.642,169.463,50.447,159.667
C03511=1019.274,262.146,367.672,169.459,50.452,159.668
C03512=1019.267,261.897,367.701,169.455,50.457,159.668
C03513=1019.261,261.649,367.730,169.450,50.463,159.668
C03514=1019.255,261.400,367.758,169.445,50.468,159.669
C03515=1019.249,261.153,367.787,169.441,50.473,159.669
C03516=1019.243,260.905,367.816,169.436,50.478,159.669
C03517=1019.237,260.656,367.844,169.432,50.483,159.670
C03518=1019.232,260.408,367.874,169.427,50.488,159.670
C03519=1019.226,260.160,367.903,169.423,50.493,159.671
C03520=1019.220,259.911,367.931,169.418,50.498,159.671
C03521=1019.213,259.663,367.959,169.414,50.503,159.671
C03522=1019.207,259.414,367.988,169.409,50.509,159.672
C03523=1019.200,259.166,368.016,169.404,50.514,159.672
C03524=1019.194,258.918,368.044,169.400,50.519,159.673
C03525=1019.188,258.670,368.073,169.395,50.525,159.673
C03526=1019.181,258.422,368.101,169.391,50.530,159.673
C03527=1019.175,258.174,368.130,169.387,50.535,159.674
C03528=1019.169,257.925,368.158,169.381,50.540,159.674
C03529=1019.163,257.677,368.186,169.377,50.546,159.675
C03530=1019.156,257.428,368.215,169.373,50.551,159.675
C03531=1019.150,257.180,368.243,169.368,50.556,159.675
C03532=1019.144,256.932,368.271,169.364,50.562,159.676
C03533=1019.138,256.684,368.300,169.359,50.567,159.676
C03534=1019.132,256.435,368.328,169.354,50.573,159.677
C03535=1019.125,256.187,368.356,169.350,50.578,159.677
C03536=1019.119,255.938,368.385,169.346,50.583,159.677
C03537=1019.113,255.690,368.413,169.341,50.588,159.678
C03538=1019.107,255.442,368.441,169.337,50.594,159.678
C03539=1019.101,255.194,368.470,169.332,50.599,159.679
C03540=1019.095,254.945,368.498,169.328,50.605,159.679
C03541=1019.088,254.697,368.526,169.323,50.610,159.679
C03542=1019.083,254.449,368.554,169.319,50.616,159.680
C03543=1019.077,254.200,368.583,169.315,50.621,159.680
C03544=1019.070,253.952,368.610,169.310,50.627,159.681
C03545=1019.064,253.703,368.639,169.306,50.632,159.681
C03546=1019.059,253.455,368.667,169.302,50.637,159.682
C03547=1019.052,253.207,368.694,169.297,50.643,159.682
C03548=1019.046,252.958,368.723,169.292,50.648,159.683
C03549=1019.040,252.710,368.752,169.288,50.654,159.683
C03550=1019.034,252.462,368.779,169.283,50.660,159.683
C03551=1019.028,252.213,368.807,169.279,50.665,159.684
C03552=1019.022,251.965,368.836,169.275,50.670,159.684
C03553=1019.016,251.717,368.863,169.270,50.676,159.685
C03554=1019.010,251.468,368.891,169.266,50.681,159.685
C03555=1019.003,251.220,368.919,169.262,50.687,159.686
C03556=1018.998,250.972,368.947,169.257,50.693,159.686
C03557=1018.992,250.723,368.975,169.252,50.698,159.687
C03558=1018.985,250.474,369.003,169.248,50.703,159.687
C03559=1018.980,250.226,369.031,169.243,50.709,159.687
C03560=1018.974,249.978,369.060,169.239,50.714,159.688
C03561=1018.967,249.729,369.087,169.235,50.720,159.688
C03562=1018.962,249.506,369.113,169.231,50.725,159.689
C03563=1018.957,249.282,369.138,169.227,50.731,159.689
C03564=1018.951,249.058,369.163,169.223,50.735,159.690
C03565=1018.946,248.834,369.188,169.219,50.740,159.690
C03566=1018.941,248.610,369.214,169.215,50.746,159.691
C03567=1018.935,248.386,369.240,169.212,50.750,159.691
C03568=1018.930,248.163,369.264,169.208,50.755,159.691
C03569=1018.925,247.939,369.289,169.204,50.761,159.692
C03570=1018.919,247.690,369.317,169.199,50.766,159.692
C03571=1018.913,247.442,369.345,169.195,50.772,159.693
C03572=1018.907,247.193,369.373,169.190,50.777,159.693
C03573=1018.901,246.946,369.401,169.186,50.783,159.694
C03574=1018.895,246.696,369.428,169.182,50.789,159.694
C03575=1018.890,246.448,369.456,169.177,50.795,159.695
C03576=1018.883,246.200,369.484,169.173,50.800,159.695
C03577=1018.878,245.952,369.512,169.170,50.806,159.696
C03578=1018.872,245.703,369.540,169.165,50.812,159.696
C03579=1018.866,245.455,369.567,169.160,50.817,159.697
C03580=1018.860,245.206,369.595,169.156,50.823,159.697
C03581=1018.855,244.958,369.623,169.152,50.829,159.698
C03582=1018.848,244.709,369.651,169.148,50.834,159.698
C03583=1018.843,244.461,369.679,169.143,50.840,159.699
C03584=1018.836,244.213,369.706,169.139,50.846,159.699
C03585=1018.831,243.964,369.734,169.135,50.852,159.700
C03586=1018.825,243.715,369.762,169.131,50.857,159.700
C03587=1018.819,243.468,369.789,169.126,50.863,159.701
C03588=1018.813,243.219,369.818,169.122,50.869,159.701
C03589=1018.807,242.971,369.844,169.118,50.875,159.702
C03590=1018.802,242.723,369.872,169.113,50.881,159.702
C03591=1018.795,242.473,369.899,169.109,50.887,159.703
C03592=1018.789,242.226,369.927,169.104,50.893,159.703
C03593=1018.784,241.976,369.954,169.101,50.899,159.704
C03594=1018.778,241.729,369.982,169.095,50.904,159.704
C03595=1018.771,241.480,370.009,169.092,50.910,159.705
C03596=1018.766,241.232,370.037,169.088,50.917,159.706
C03597=1018.760,240.983,370.063,169.083,50.922,159.706
C03598=1018.753,240.735,370.091,169.079,50.928,159.707
C03599=1018.748,240.486,370.118,169.074,50.934,159.707
C03600=1018.742,240.238,370.146,169.071,50.940,159.708
C03601=1018.736,239.989,370.173,169.067,50.946,159.709
C03602=1018.731,239.741,370.201,169.062,50.952,159.709
C03603=1018.724,239.492,370.228,169.058,50.958,159.710
C03604=1018.718,239.244,370.255,169.053,50.965,159.710
C03605=1018.713,238.996,370.282,169.049,50.970,159.711
C03606=1018.707,238.747,370.309,169.045,50.976,159.711
C03607=1018.701,238.499,370.337,169.041,50.983,159.712
C03608=1018.694,238.250,370.364,169.036,50.989,159.712
C03609=1018.688,238.002,370.390,169.033,50.995,159.713
C03610=1018.683,237.753,370.417,169.028,51.001,159.714
C03611=1018.676,237.505,370.445,169.024,51.007,159.714
C03612=1018.670,237.256,370.471,169.019,51.013,159.715
C03613=1018.664,237.008,370.498,169.016,51.020,159.715
C03614=1018.658,236.759,370.525,169.011,51.026,159.716
C03615=1018.652,236.511,370.552,169.007,51.032,159.717
C03616=1018.646,236.263,370.579,169.004,51.038,159.717
C03617=1018.641,236.013,370.607,168.999,51.045,159.718
C03618=1018.635,235.765,370.633,168.994,51.051,159.719
C03619=1018.629,235.517,370.660,168.991,51.057,159.719
C03620=1018.623,235.268,370.687,168.985,51.063,159.720
C03621=1018.617,235.019,370.714,168.982,51.069,159.720
C03622=1018.611,234.792,370.738,168.978,51.075,159.721
C03623=1018.605,234.565,370.763,168.974,51.081,159.721
C03624=1018.600,234.338,370.787,168.970,51.087,159.722
C03625=1018.595,234.111,370.811,168.966,51.092,159.723
C03626=1018.590,233.885,370.836,168.963,51.098,159.723
C03627=1018.584,233.657,370.860,168.959,51.104,159.724
C03628=1018.578,233.430,370.885,168.955,51.110,159.724
C03629=1018.573,233.203,370.910,168.951,51.116,159.725
C03630=1018.567,232.954,370.936,168.948,51.122,159.726
C03631=1018.562,232.706,370.963,168.943,51.129,159.726
C03632=1018.555,232.457,370.990,168.939,51.135,159.727
C03633=1018.550,232.209,371.017,168.935,51.141,159.728
C03634=1018.544,231.960,371.043,168.931,51.147,159.728
C03635=1018.538,231.712,371.070,168.926,51.154,159.729
C03636=1018.532,231.464,371.097,168.922,51.160,159.729
C03637=1018.526,231.214,371.123,168.918,51.166,159.730
C03638=1018.520,230.966,371.150,168.913,51.173,159.731
C03639=1018.515,230.717,371.176,168.910,51.180,159.731
C03640=1018.509,230.469,371.203,168.906,51.186,159.732
